LIN {X 0,Y 481.377,Z 604.114,A -85,B 0,C 180,E1 -6920.97,E2 -6920.97} C_VEL
LIN {X 0,Y 481.208,Z 611.494,A -85,B 0,C 180,E1 -6922.236,E2 -6922.236} C_VEL
LIN {X 0,Y 481.101,Z 618.078,A -85,B 0,C 180,E1 -6923.67,E2 -6923.67} C_VEL
LIN {X 0,Y 481.076,Z 622.704,A -85,B 0,C 180,E1 -6924.971,E2 -6924.971} C_VEL
LIN {X 0,Y 481.102,Z 625.077,A -85,B 0,C 180,E1 -6925.811,E2 -6925.811} C_VEL
LIN {X 0,Y 481.058,Z 626.993,A -85,B 0,C 180,E1 -6926.65,E2 -6926.65} C_VEL
LIN {X 0,Y 481.036,Z 628.433,A -85,B 0,C 180,E1 -6927.488,E2 -6927.488} C_VEL
LIN {X 0,Y 481.062,Z 630.096,A -85,B 0,C 180,E1 -6929.163,E2 -6929.163} C_VEL
LIN {X 0,Y 481.049,Z 630.319,A -85,B 0,C 180,E1 -6930,E2 -6930} C_VEL
LIN {X 0,Y 481.062,Z 630.101,A -85,B 0,C 180,E1 -6930.837,E2 -6930.837} C_VEL
LIN {X 0,Y 481.035,Z 628.45,A -85,B 0,C 180,E1 -6932.512,E2 -6932.512} C_VEL
LIN {X 0,Y 481.056,Z 627.015,A -85,B 0,C 180,E1 -6933.35,E2 -6933.35} C_VEL
LIN {X 0,Y 481.046,Z 623.991,A -85,B 0,C 180,E1 -6934.609,E2 -6934.609} C_VEL
LIN {X 0,Y 481.125,Z 619.912,A -85,B 0,C 180,E1 -6935.869,E2 -6935.869} C_VEL
LIN {X 0,Y 481.153,Z 613.626,A -85,B 0,C 180,E1 -6937.343,E2 -6937.343} C_VEL
LIN {X 0,Y 481.309,Z 606.787,A -85,B 0,C 180,E1 -6938.608,E2 -6938.608} C_VEL
LIN {X 0,Y 481.523,Z 598.317,A -85,B 0,C 180,E1 -6939.875,E2 -6939.875} C_VEL
LIN {X 0,Y 481.865,Z 589.664,A -85,B 0,C 180,E1 -6940.93,E2 -6940.93} C_VEL
LIN {X 0,Y 482.304,Z 579.305,A -85,B 0,C 180,E1 -6941.958,E2 -6941.958} C_VEL
LIN {X 0,Y 482.668,Z 568.475,A -85,B 0,C 180,E1 -6942.829,E2 -6942.829} C_VEL
LIN {X 0,Y 483.085,Z 556.965,A -85,B 0,C 180,E1 -6943.567,E2 -6943.567} C_VEL
LIN {X 0,Y 483.501,Z 545.184,A -85,B 0,C 180,E1 -6944.145,E2 -6944.145} C_VEL
LIN {X 0,Y 483.517,Z 538.3,A -85,B 0,C 180,E1 -6944.413,E2 -6944.413} C_VEL
LIN {X 0,Y 482.293,Z 527.392,A -85,B 0,C 180,E1 -6944.774,E2 -6944.774} C_VEL
LIN {X 0,Y 481.44,Z 518.405,A -85,B 0,C 180,E1 -6944.99,E2 -6944.99} C_VEL
LIN {X 0,Y 481.705,Z 503.738,A -85,B 0,C 180,E1 -6948.169,E2 -6948.169} C_VEL
LIN {X 0,Y 481.993,Z 488.984,A -85,B 0,C 180,E1 -6951.378,E2 -6951.378} C_VEL
LIN {X 0,Y 482.327,Z 474.573,A -85,B 0,C 180,E1 -6954.536,E2 -6954.536} C_VEL
LIN {X 0,Y 482.614,Z 461.951,A -85,B 0,C 180,E1 -6957.339,E2 -6957.339} C_VEL
LIN {X 0,Y 482.979,Z 449.607,A -85,B 0,C 180,E1 -6960.134,E2 -6960.134} C_VEL
LIN {X 0,Y 483.414,Z 436.079,A -85,B 0,C 180,E1 -6963.286,E2 -6963.286} C_VEL
LIN {X 0,Y 483.897,Z 423.674,A -85,B 0,C 180,E1 -6966.288,E2 -6966.288} C_VEL
LIN {X 0,Y 482.493,Z 415.613,A -85,B 0,C 180,E1 -6968.425,E2 -6968.425} C_VEL
LIN {X 0,Y 481.728,Z 411.479,A -85,B 0,C 180,E1 -6969.609,E2 -6969.609} C_VEL
LIN {X 0,Y 481.644,Z 411.493,A -85,B 0,C 180,E1 -6973.148,E2 -6973.148} C_VEL
LIN {X 0,Y 481.66,Z 411.49,A -85,B 0,C 180,E1 -6975.641,E2 -6975.641} C_VEL
LIN {X 0,Y 481.664,Z 411.488,A -85,B 0,C 180,E1 -6978.959,E2 -6978.959} C_VEL
LIN {X 0,Y 481.658,Z 411.49,A -85,B 0,C 180,E1 -6981.992,E2 -6981.992} C_VEL
LIN {X 0,Y 481.693,Z 411.483,A -85,B 0,C 180,E1 -6985.318,E2 -6985.318} C_VEL
LIN {X 0,Y 481.646,Z 411.491,A -85,B 0,C 180,E1 -6988.312,E2 -6988.312} C_VEL
LIN {X 0,Y 481.702,Z 411.482,A -85,B 0,C 180,E1 -6991.219,E2 -6991.219} C_VEL
LIN {X 0,Y 481.708,Z 411.484,A -85,B 0,C 180,E1 -6994.043,E2 -6994.043} C_VEL
LIN {X 0,Y 481.676,Z 411.486,A -85,B 0,C 180,E1 -6996.812,E2 -6996.812} C_VEL
LIN {X 0,Y 481.699,Z 411.483,A -85,B 0,C 180,E1 -6999.503,E2 -6999.503} C_VEL
LIN {X 0,Y 481.709,Z 411.484,A -85,B 0,C 180,E1 -7002.159,E2 -7002.159} C_VEL
LIN {X 0,Y 481.744,Z 411.479,A -85,B 0,C 180,E1 -7004.776,E2 -7004.776} C_VEL
LIN {X 0,Y 481.797,Z 411.474,A -85,B 0,C 180,E1 -7008.216,E2 -7008.216} C_VEL
LIN {X 0,Y 481.742,Z 411.479,A -85,B 0,C 180,E1 -7011.611,E2 -7011.611} C_VEL
LIN {X 0,Y 481.819,Z 411.47,A -85,B 0,C 180,E1 -7014.14,E2 -7014.14} C_VEL
LIN {X 0,Y 481.932,Z 411.455,A -85,B 0,C 180,E1 -7017.493,E2 -7017.493} C_VEL
LIN {X 0,Y 481.909,Z 411.457,A -85,B 0,C 180,E1 -7020.836,E2 -7020.836} C_VEL
LIN {X 0,Y 481.929,Z 411.455,A -85,B 0,C 180,E1 -7022.508,E2 -7022.508} C_VEL
LIN {X 0,Y 481.818,Z 411.471,A -85,B 0,C 180,E1 -7025.861,E2 -7025.861} C_VEL
LIN {X 0,Y 481.766,Z 411.476,A -85,B 0,C 180,E1 -7028.388,E2 -7028.388} C_VEL
LIN {X 0,Y 481.753,Z 411.478,A -85,B 0,C 180,E1 -7031.785,E2 -7031.785} C_VEL
LIN {X 0,Y 481.745,Z 411.477,A -85,B 0,C 180,E1 -7035.224,E2 -7035.224} C_VEL
LIN {X 0,Y 481.715,Z 411.481,A -85,B 0,C 180,E1 -7038.722,E2 -7038.722} C_VEL
LIN {X 0,Y 481.65,Z 411.49,A -85,B 0,C 180,E1 -7041.395,E2 -7041.395} C_VEL
LIN {X 0,Y 481.68,Z 411.488,A -85,B 0,C 180,E1 -7044.113,E2 -7044.113} C_VEL
LIN {X 0,Y 481.749,Z 411.477,A -85,B 0,C 180,E1 -7047.139,E2 -7047.139} C_VEL
LIN {X 0,Y 481.681,Z 411.488,A -85,B 0,C 180,E1 -7049.741,E2 -7049.741} C_VEL
LIN {X 0,Y 481.675,Z 411.486,A -85,B 0,C 180,E1 -7052.674,E2 -7052.674} C_VEL
LIN {X 0,Y 481.645,Z 411.492,A -85,B 0,C 180,E1 -7055.709,E2 -7055.709} C_VEL
LIN {X 0,Y 481.673,Z 411.486,A -85,B 0,C 180,E1 -7058.859,E2 -7058.859} C_VEL
LIN {X 0,Y 481.665,Z 411.489,A -85,B 0,C 180,E1 -7061.914,E2 -7061.914} C_VEL
LIN {X 0,Y 481.663,Z 411.489,A -85,B 0,C 180,E1 -7064.457,E2 -7064.457} C_VEL
LIN {X 0,Y 481.657,Z 411.492,A -85,B 0,C 180,E1 -7067.84,E2 -7067.84} C_VEL
LIN {X 0,Y 481.684,Z 411.485,A -85,B 0,C 180,E1 -7070.651,E2 -7070.651} C_VEL
LIN {X 0,Y 481.634,Z 411.493,A -85,B 0,C 180,E1 -7073.376,E2 -7073.376} C_VEL
LIN {X 0,Y 481.713,Z 411.483,A -85,B 0,C 180,E1 -7076.33,E2 -7076.33} C_VEL
LIN {X 0,Y 481.663,Z 411.489,A -85,B 0,C 180,E1 -7079.416,E2 -7079.416} C_VEL
LIN {X 0,Y 481.705,Z 411.483,A -85,B 0,C 180,E1 -7082.168,E2 -7082.168} C_VEL
LIN {X 0,Y 481.721,Z 411.48,A -85,B 0,C 180,E1 -7084.97,E2 -7084.97} C_VEL
LIN {X 0,Y 481.64,Z 411.49,A -85,B 0,C 180,E1 -7087.985,E2 -7087.985} C_VEL
LIN {X 0,Y 480.972,Z 411.574,A -85,B 0,C 180,E1 -7088.683,E2 -7088.683} C_VEL
LIN {X 0,Y 478.146,Z 411.927,A -85,B 0,C 180,E1 -7089.817,E2 -7089.817} C_VEL
LIN {X 0,Y 475.762,Z 412.224,A -85,B 0,C 180,E1 -7090.732,E2 -7090.732} C_VEL
LIN {X 0,Y 474.742,Z 412.351,A -85,B 0,C 180,E1 -7091.437,E2 -7091.437} C_VEL
LIN {X 0,Y 474.66,Z 412.361,A -85,B 0,C 180,E1 -7091.676,E2 -7091.676} C_VEL
LIN {X 0,Y 474.705,Z 412.355,A -85,B 0,C 180,E1 -7094.545,E2 -7094.545} C_VEL
LIN {X 0,Y 474.709,Z 412.354,A -85,B 0,C 180,E1 -7098.038,E2 -7098.038} C_VEL
LIN {X 0,Y 474.762,Z 412.348,A -85,B 0,C 180,E1 -7098.689,E2 -7098.689} C_VEL
LIN {X 0,Y 477.209,Z 421.926,A -85,B 0,C 180,E1 -7099.285,E2 -7099.285} C_VEL
LIN {X 0,Y 476.901,Z 433.183,A -85,B 0,C 180,E1 -7100.029,E2 -7100.029} C_VEL
LIN {X 0,Y 476.389,Z 444.579,A -85,B 0,C 180,E1 -7100.982,E2 -7100.982} C_VEL
LIN {X 0,Y 475.996,Z 453.528,A -85,B 0,C 180,E1 -7101.913,E2 -7101.913} C_VEL
LIN {X 0,Y 475.625,Z 462.093,A -85,B 0,C 180,E1 -7102.998,E2 -7102.998} C_VEL
LIN {X 0,Y 475.251,Z 470.197,A -85,B 0,C 180,E1 -7104.271,E2 -7104.271} C_VEL
LIN {X 0,Y 474.95,Z 475.754,A -85,B 0,C 180,E1 -7105.332,E2 -7105.332} C_VEL
LIN {X 0,Y 474.707,Z 481.159,A -85,B 0,C 180,E1 -7106.605,E2 -7106.605} C_VEL
LIN {X 0,Y 474.572,Z 485.4,A -85,B 0,C 180,E1 -7107.878,E2 -7107.878} C_VEL
LIN {X 0,Y 474.352,Z 488.628,A -85,B 0,C 180,E1 -7109.151,E2 -7109.151} C_VEL
LIN {X 0,Y 474.295,Z 490.225,A -85,B 0,C 180,E1 -7110,E2 -7110} C_VEL
LIN {X 0,Y 474.172,Z 491.447,A -85,B 0,C 180,E1 -7110.849,E2 -7110.849} C_VEL
LIN {X 0,Y 474.232,Z 492.256,A -85,B 0,C 180,E1 -7111.699,E2 -7111.699} C_VEL
LIN {X 0,Y 474.206,Z 492.692,A -85,B 0,C 180,E1 -7113.399,E2 -7113.399} C_VEL
LIN {X 0,Y 474.321,Z 491.624,A -85,B 0,C 180,E1 -7115.101,E2 -7115.101} C_VEL
LIN {X 0,Y 474.401,Z 488.934,A -85,B 0,C 180,E1 -7116.807,E2 -7116.807} C_VEL
LIN {X 0,Y 474.522,Z 485.822,A -85,B 0,C 180,E1 -7118.089,E2 -7118.089} C_VEL
LIN {X 0,Y 474.749,Z 481.653,A -85,B 0,C 180,E1 -7119.372,E2 -7119.372} C_VEL
LIN {X 0,Y 475.063,Z 475.32,A -85,B 0,C 180,E1 -7120.873,E2 -7120.873} C_VEL
LIN {X 0,Y 475.337,Z 468.074,A -85,B 0,C 180,E1 -7122.206,E2 -7122.206} C_VEL
LIN {X 0,Y 475.767,Z 459.593,A -85,B 0,C 180,E1 -7123.454,E2 -7123.454} C_VEL
LIN {X 0,Y 476.167,Z 450.586,A -85,B 0,C 180,E1 -7124.532,E2 -7124.532} C_VEL
LIN {X 0,Y 476.623,Z 440.519,A -85,B 0,C 180,E1 -7125.502,E2 -7125.502} C_VEL
LIN {X 0,Y 477.01,Z 429.745,A -85,B 0,C 180,E1 -7126.335,E2 -7126.335} C_VEL
LIN {X 0,Y 477.127,Z 420.99,A -85,B 0,C 180,E1 -7126.89,E2 -7126.89} C_VEL
LIN {X 0,Y 474.656,Z 412.36,A -85,B 0,C 180,E1 -7127.448,E2 -7127.448} C_VEL
LIN {X 0,Y 474.659,Z 412.361,A -85,B 0,C 180,E1 -7129.91,E2 -7129.91} C_VEL
LIN {X 0,Y 474.64,Z 412.357,A -85,B 0,C 180,E1 -7133.358,E2 -7133.358} C_VEL
LIN {X 0,Y 474.66,Z 412.362,A -85,B 0,C 180,E1 -7136.372,E2 -7136.372} C_VEL
LIN {X 0,Y 474.626,Z 412.359,A -85,B 0,C 180,E1 -7139.252,E2 -7139.252} C_VEL
LIN {X 0,Y 474.62,Z 412.365,A -85,B 0,C 180,E1 -7142.431,E2 -7142.431} C_VEL
LIN {X 0,Y 474.624,Z 412.36,A -85,B 0,C 180,E1 -7145.47,E2 -7145.47} C_VEL
LIN {X 0,Y 474.617,Z 412.364,A -85,B 0,C 180,E1 -7148.457,E2 -7148.457} C_VEL
LIN {X 0,Y 474.632,Z 412.358,A -85,B 0,C 180,E1 -7150.959,E2 -7150.959} C_VEL
LIN {X 0,Y 474.614,Z 412.369,A -85,B 0,C 180,E1 -7154.105,E2 -7154.105} C_VEL
LIN {X 0,Y 474.62,Z 412.359,A -85,B 0,C 180,E1 -7157.066,E2 -7157.066} C_VEL
LIN {X 0,Y 474.649,Z 412.358,A -85,B 0,C 180,E1 -7160.454,E2 -7160.454} C_VEL
LIN {X 0,Y 474.593,Z 412.367,A -85,B 0,C 180,E1 -7163.676,E2 -7163.676} C_VEL
LIN {X 0,Y 474.647,Z 412.356,A -85,B 0,C 180,E1 -7166.78,E2 -7166.78} C_VEL
LIN {X 0,Y 474.61,Z 412.367,A -85,B 0,C 180,E1 -7169.77,E2 -7169.77} C_VEL
LIN {X 0,Y 474.702,Z 412.349,A -85,B 0,C 180,E1 -7172.68,E2 -7172.68} C_VEL
LIN {X 0,Y 474.645,Z 412.36,A -85,B 0,C 180,E1 -7175.506,E2 -7175.506} C_VEL
LIN {X 0,Y 474.675,Z 412.354,A -85,B 0,C 180,E1 -7179.185,E2 -7179.185} C_VEL
LIN {X 0,Y 474.651,Z 412.362,A -85,B 0,C 180,E1 -7181.884,E2 -7181.884} C_VEL
LIN {X 0,Y 474.704,Z 412.349,A -85,B 0,C 180,E1 -7184.544,E2 -7184.544} C_VEL
LIN {X 0,Y 474.662,Z 412.358,A -85,B 0,C 180,E1 -7186.874,E2 -7186.874} C_VEL
LIN {X 0,Y 476.753,Z 420.106,A -85,B 0,C 180,E1 -7187.367,E2 -7187.367} C_VEL
LIN {X 0,Y 476.502,Z 430.082,A -85,B 0,C 180,E1 -7188.007,E2 -7188.007} C_VEL
LIN {X 0,Y 476.131,Z 441.708,A -85,B 0,C 180,E1 -7188.937,E2 -7188.937} C_VEL
LIN {X 0,Y 475.81,Z 450.358,A -85,B 0,C 180,E1 -7189.79,E2 -7189.79} C_VEL
LIN {X 0,Y 475.421,Z 459.298,A -85,B 0,C 180,E1 -7190.856,E2 -7190.856} C_VEL
LIN {X 0,Y 475.084,Z 468.019,A -85,B 0,C 180,E1 -7192.135,E2 -7192.135} C_VEL
LIN {X 0,Y 474.872,Z 475.039,A -85,B 0,C 180,E1 -7193.414,E2 -7193.414} C_VEL
LIN {X 0,Y 474.479,Z 481.448,A -85,B 0,C 180,E1 -7194.901,E2 -7194.901} C_VEL
LIN {X 0,Y 474.487,Z 485.65,A -85,B 0,C 180,E1 -7196.178,E2 -7196.178} C_VEL
LIN {X 0,Y 474.218,Z 488.842,A -85,B 0,C 180,E1 -7197.452,E2 -7197.452} C_VEL
LIN {X 0,Y 474.242,Z 490.427,A -85,B 0,C 180,E1 -7198.301,E2 -7198.301} C_VEL
LIN {X 0,Y 474.17,Z 491.584,A -85,B 0,C 180,E1 -7199.151,E2 -7199.151} C_VEL
LIN {X 0,Y 474.167,Z 492.694,A -85,B 0,C 180,E1 -7200.849,E2 -7200.849} C_VEL
LIN {X 0,Y 474.232,Z 492.669,A -85,B 0,C 180,E1 -7201.698,E2 -7201.698} C_VEL
LIN {X 0,Y 474.263,Z 491.378,A -85,B 0,C 180,E1 -7203.398,E2 -7203.398} C_VEL
LIN {X 0,Y 474.329,Z 490.156,A -85,B 0,C 180,E1 -7204.248,E2 -7204.248} C_VEL
LIN {X 0,Y 474.483,Z 487.49,A -85,B 0,C 180,E1 -7205.525,E2 -7205.525} C_VEL
LIN {X 0,Y 474.665,Z 483.805,A -85,B 0,C 180,E1 -7206.803,E2 -7206.803} C_VEL
LIN {X 0,Y 474.832,Z 478.985,A -85,B 0,C 180,E1 -7208.083,E2 -7208.083} C_VEL
LIN {X 0,Y 475.145,Z 472.826,A -85,B 0,C 180,E1 -7209.364,E2 -7209.364} C_VEL
LIN {X 0,Y 475.462,Z 465.142,A -85,B 0,C 180,E1 -7210.648,E2 -7210.648} C_VEL
LIN {X 0,Y 475.809,Z 457.258,A -85,B 0,C 180,E1 -7211.718,E2 -7211.718} C_VEL
LIN {X 0,Y 476.148,Z 447.587,A -85,B 0,C 180,E1 -7212.791,E2 -7212.791} C_VEL
LIN {X 0,Y 476.651,Z 436.734,A -85,B 0,C 180,E1 -7213.754,E2 -7213.754} C_VEL
LIN {X 0,Y 477.028,Z 426.184,A -85,B 0,C 180,E1 -7214.505,E2 -7214.505} C_VEL
LIN {X 0,Y 476.99,Z 420.79,A -85,B 0,C 180,E1 -7214.833,E2 -7214.833} C_VEL
LIN {X 0,Y 474.697,Z 412.357,A -85,B 0,C 180,E1 -7215.373,E2 -7215.373} C_VEL
LIN {X 0,Y 474.663,Z 412.366,A -85,B 0,C 180,E1 -7218.629,E2 -7218.629} C_VEL
LIN {X 0,Y 474.639,Z 412.367,A -85,B 0,C 180,E1 -7221.116,E2 -7221.116} C_VEL
LIN {X 0,Y 474.644,Z 412.363,A -85,B 0,C 180,E1 -7224.494,E2 -7224.494} C_VEL
LIN {X 0,Y 474.703,Z 412.355,A -85,B 0,C 180,E1 -7227.338,E2 -7227.338} C_VEL
LIN {X 0,Y 474.608,Z 412.367,A -85,B 0,C 180,E1 -7230.81,E2 -7230.81} C_VEL
LIN {X 0,Y 474.641,Z 412.363,A -85,B 0,C 180,E1 -7233.984,E2 -7233.984} C_VEL
LIN {X 0,Y 474.575,Z 412.372,A -85,B 0,C 180,E1 -7236.899,E2 -7236.899} C_VEL
LIN {X 0,Y 474.63,Z 412.364,A -85,B 0,C 180,E1 -7239.647,E2 -7239.647} C_VEL
LIN {X 0,Y 474.618,Z 412.366,A -85,B 0,C 180,E1 -7242.934,E2 -7242.934} C_VEL
LIN {X 0,Y 474.612,Z 412.364,A -85,B 0,C 180,E1 -7245.895,E2 -7245.895} C_VEL
LIN {X 0,Y 474.631,Z 412.364,A -85,B 0,C 180,E1 -7249.041,E2 -7249.041} C_VEL
LIN {X 0,Y 474.67,Z 412.558,A -85,B 0,C 180,E1 -7249.868,E2 -7249.868} C_VEL
LIN {X 0,Y 476.752,Z 422.929,A -85,B 0,C 180,E1 -7252.814,E2 -7252.814} C_VEL
LIN {X 0,Y 477.156,Z 426.977,A -85,B 0,C 180,E1 -7253.902,E2 -7253.902} C_VEL
LIN {X 0,Y 476.36,Z 441.74,A -85,B 0,C 180,E1 -7257.572,E2 -7257.572} C_VEL
LIN {X 0,Y 475.905,Z 454.457,A -85,B 0,C 180,E1 -7260.609,E2 -7260.609} C_VEL
LIN {X 0,Y 475.492,Z 467.701,A -85,B 0,C 180,E1 -7263.678,E2 -7263.678} C_VEL
LIN {X 0,Y 475.158,Z 480.12,A -85,B 0,C 180,E1 -7266.497,E2 -7266.497} C_VEL
LIN {X 0,Y 474.78,Z 494.181,A -85,B 0,C 180,E1 -7269.643,E2 -7269.643} C_VEL
LIN {X 0,Y 474.542,Z 508.253,A -85,B 0,C 180,E1 -7272.77,E2 -7272.77} C_VEL
LIN {X 0,Y 474.368,Z 517.338,A -85,B 0,C 180,E1 -7274.781,E2 -7274.781} C_VEL
LIN {X 0,Y 475.741,Z 532.276,A -85,B 0,C 180,E1 -7275.182,E2 -7275.182} C_VEL
LIN {X 0,Y 476.7,Z 541.484,A -85,B 0,C 180,E1 -7275.539,E2 -7275.539} C_VEL
LIN {X 0,Y 476.207,Z 553.915,A -85,B 0,C 180,E1 -7276.124,E2 -7276.124} C_VEL
LIN {X 0,Y 475.712,Z 565.91,A -85,B 0,C 180,E1 -7276.871,E2 -7276.871} C_VEL
LIN {X 0,Y 475.293,Z 576.474,A -85,B 0,C 180,E1 -7277.707,E2 -7277.707} C_VEL
LIN {X 0,Y 474.861,Z 586.571,A -85,B 0,C 180,E1 -7278.691,E2 -7278.691} C_VEL
LIN {X 0,Y 474.527,Z 595.599,A -85,B 0,C 180,E1 -7279.762,E2 -7279.762} C_VEL
LIN {X 0,Y 474.265,Z 604.436,A -85,B 0,C 180,E1 -7281.048,E2 -7281.048} C_VEL
LIN {X 0,Y 474.108,Z 611.516,A -85,B 0,C 180,E1 -7282.333,E2 -7282.333} C_VEL
LIN {X 0,Y 474.037,Z 617.39,A -85,B 0,C 180,E1 -7283.663,E2 -7283.663} C_VEL
LIN {X 0,Y 474.03,Z 621.682,A -85,B 0,C 180,E1 -7284.896,E2 -7284.896} C_VEL
LIN {X 0,Y 474.036,Z 624.054,A -85,B 0,C 180,E1 -7285.749,E2 -7285.749} C_VEL
LIN {X 0,Y 474.013,Z 625.974,A -85,B 0,C 180,E1 -7286.6,E2 -7286.6} C_VEL
LIN {X 0,Y 473.997,Z 627.416,A -85,B 0,C 180,E1 -7287.45,E2 -7287.45} C_VEL
LIN {X 0,Y 474.051,Z 629.086,A -85,B 0,C 180,E1 -7289.15,E2 -7289.15} C_VEL
LIN {X 0,Y 474.036,Z 629.31,A -85,B 0,C 180,E1 -7290,E2 -7290} C_VEL
LIN {X 0,Y 474.05,Z 629.092,A -85,B 0,C 180,E1 -7290.849,E2 -7290.849} C_VEL
LIN {X 0,Y 473.995,Z 627.437,A -85,B 0,C 180,E1 -7292.549,E2 -7292.549} C_VEL
LIN {X 0,Y 474.01,Z 626,A -85,B 0,C 180,E1 -7293.4,E2 -7293.4} C_VEL
LIN {X 0,Y 474.001,Z 622.976,A -85,B 0,C 180,E1 -7294.677,E2 -7294.677} C_VEL
LIN {X 0,Y 474.06,Z 618.892,A -85,B 0,C 180,E1 -7295.956,E2 -7295.956} C_VEL
LIN {X 0,Y 474.099,Z 612.606,A -85,B 0,C 180,E1 -7297.453,E2 -7297.453} C_VEL
LIN {X 0,Y 474.236,Z 605.761,A -85,B 0,C 180,E1 -7298.737,E2 -7298.737} C_VEL
LIN {X 0,Y 474.476,Z 597.292,A -85,B 0,C 180,E1 -7300.023,E2 -7300.023} C_VEL
LIN {X 0,Y 474.825,Z 588.636,A -85,B 0,C 180,E1 -7301.094,E2 -7301.094} C_VEL
LIN {X 0,Y 475.291,Z 578.561,A -85,B 0,C 180,E1 -7302.111,E2 -7302.111} C_VEL
LIN {X 0,Y 475.623,Z 568.892,A -85,B 0,C 180,E1 -7302.914,E2 -7302.914} C_VEL
LIN {X 0,Y 476.068,Z 557.722,A -85,B 0,C 180,E1 -7303.662,E2 -7303.662} C_VEL
LIN {X 0,Y 476.527,Z 545.375,A -85,B 0,C 180,E1 -7304.302,E2 -7304.302} C_VEL
LIN {X 0,Y 476.475,Z 538.387,A -85,B 0,C 180,E1 -7304.59,E2 -7304.59} C_VEL
LIN {X 0,Y 475.375,Z 527.969,A -85,B 0,C 180,E1 -7304.953,E2 -7304.953} C_VEL
LIN {X 0,Y 474.368,Z 517.419,A -85,B 0,C 180,E1 -7305.219,E2 -7305.219} C_VEL
LIN {X 0,Y 474.635,Z 503.154,A -85,B 0,C 180,E1 -7308.367,E2 -7308.367} C_VEL
LIN {X 0,Y 474.953,Z 488.049,A -85,B 0,C 180,E1 -7311.711,E2 -7311.711} C_VEL
LIN {X 0,Y 475.318,Z 473.658,A -85,B 0,C 180,E1 -7314.923,E2 -7314.923} C_VEL
LIN {X 0,Y 475.694,Z 459.14,A -85,B 0,C 180,E1 -7318.214,E2 -7318.214} C_VEL
LIN {X 0,Y 476.092,Z 446.662,A -85,B 0,C 180,E1 -7321.109,E2 -7321.109} C_VEL
LIN {X 0,Y 476.603,Z 433.186,A -85,B 0,C 180,E1 -7324.332,E2 -7324.332} C_VEL
LIN {X 0,Y 476.938,Z 424.934,A -85,B 0,C 180,E1 -7326.376,E2 -7326.376} C_VEL
LIN {X 0,Y 475.59,Z 417.265,A -85,B 0,C 180,E1 -7328.445,E2 -7328.445} C_VEL
LIN {X 0,Y 474.696,Z 412.356,A -85,B 0,C 180,E1 -7329.849,E2 -7329.849} C_VEL
LIN {X 0,Y 474.616,Z 412.369,A -85,B 0,C 180,E1 -7332.934,E2 -7332.934} C_VEL
LIN {X 0,Y 474.616,Z 412.368,A -85,B 0,C 180,E1 -7335.896,E2 -7335.896} C_VEL
LIN {X 0,Y 474.633,Z 412.363,A -85,B 0,C 180,E1 -7339.04,E2 -7339.04} C_VEL
LIN {X 0,Y 474.612,Z 412.367,A -85,B 0,C 180,E1 -7341.704,E2 -7341.704} C_VEL
LIN {X 0,Y 474.63,Z 412.364,A -85,B 0,C 180,E1 -7344.726,E2 -7344.726} C_VEL
LIN {X 0,Y 474.636,Z 412.364,A -85,B 0,C 180,E1 -7347.788,E2 -7347.788} C_VEL
LIN {X 0,Y 474.625,Z 412.365,A -85,B 0,C 180,E1 -7350.884,E2 -7350.884} C_VEL
LIN {X 0,Y 474.668,Z 412.36,A -85,B 0,C 180,E1 -7353.629,E2 -7353.629} C_VEL
LIN {X 0,Y 474.637,Z 412.363,A -85,B 0,C 180,E1 -7356.641,E2 -7356.641} C_VEL
LIN {X 0,Y 474.658,Z 412.362,A -85,B 0,C 180,E1 -7360.09,E2 -7360.09} C_VEL
LIN {X 0,Y 474.653,Z 412.361,A -85,B 0,C 180,E1 -7362.775,E2 -7362.775} C_VEL
LIN {X 0,Y 474.65,Z 412.362,A -85,B 0,C 180,E1 -7365.421,E2 -7365.421} C_VEL
LIN {X 0,Y 474.741,Z 412.352,A -85,B 0,C 180,E1 -7368.039,E2 -7368.039} C_VEL
LIN {X 0,Y 474.714,Z 412.353,A -85,B 0,C 180,E1 -7371.486,E2 -7371.486} C_VEL
LIN {X 0,Y 474.781,Z 412.347,A -85,B 0,C 180,E1 -7374.053,E2 -7374.053} C_VEL
LIN {X 0,Y 474.898,Z 412.331,A -85,B 0,C 180,E1 -7377.456,E2 -7377.456} C_VEL
LIN {X 0,Y 474.914,Z 412.33,A -85,B 0,C 180,E1 -7380,E2 -7380} C_VEL
LIN {X 0,Y 474.895,Z 412.331,A -85,B 0,C 180,E1 -7382.545,E2 -7382.545} C_VEL
LIN {X 0,Y 474.781,Z 412.347,A -85,B 0,C 180,E1 -7385.948,E2 -7385.948} C_VEL
LIN {X 0,Y 474.731,Z 412.353,A -85,B 0,C 180,E1 -7388.514,E2 -7388.514} C_VEL
LIN {X 0,Y 474.707,Z 412.357,A -85,B 0,C 180,E1 -7391.963,E2 -7391.963} C_VEL
LIN {X 0,Y 474.702,Z 412.356,A -85,B 0,C 180,E1 -7395.456,E2 -7395.456} C_VEL
LIN {X 0,Y 474.668,Z 412.358,A -85,B 0,C 180,E1 -7399.01,E2 -7399.01} C_VEL
LIN {X 0,Y 474.593,Z 412.37,A -85,B 0,C 180,E1 -7401.729,E2 -7401.729} C_VEL
LIN {X 0,Y 474.662,Z 412.36,A -85,B 0,C 180,E1 -7404.493,E2 -7404.493} C_VEL
LIN {X 0,Y 474.701,Z 412.355,A -85,B 0,C 180,E1 -7407.339,E2 -7407.339} C_VEL
LIN {X 0,Y 474.607,Z 412.366,A -85,B 0,C 180,E1 -7410.81,E2 -7410.81} C_VEL
LIN {X 0,Y 474.641,Z 412.364,A -85,B 0,C 180,E1 -7413.984,E2 -7413.984} C_VEL
LIN {X 0,Y 474.577,Z 412.37,A -85,B 0,C 180,E1 -7416.9,E2 -7416.9} C_VEL
LIN {X 0,Y 474.63,Z 412.365,A -85,B 0,C 180,E1 -7419.648,E2 -7419.648} C_VEL
LIN {X 0,Y 474.638,Z 412.362,A -85,B 0,C 180,E1 -7422.932,E2 -7422.932} C_VEL
LIN {X 0,Y 474.618,Z 412.367,A -85,B 0,C 180,E1 -7425.896,E2 -7425.896} C_VEL
LIN {X 0,Y 474.635,Z 412.363,A -85,B 0,C 180,E1 -7429.04,E2 -7429.04} C_VEL
LIN {X 0,Y 474.614,Z 412.367,A -85,B 0,C 180,E1 -7431.704,E2 -7431.704} C_VEL
LIN {X 0,Y 474.633,Z 412.362,A -85,B 0,C 180,E1 -7434.726,E2 -7434.726} C_VEL
LIN {X 0,Y 474.642,Z 412.364,A -85,B 0,C 180,E1 -7437.788,E2 -7437.788} C_VEL
LIN {X 0,Y 474.635,Z 412.363,A -85,B 0,C 180,E1 -7440.883,E2 -7440.883} C_VEL
LIN {X 0,Y 474.665,Z 412.361,A -85,B 0,C 180,E1 -7443.629,E2 -7443.629} C_VEL
LIN {X 0,Y 474.639,Z 412.361,A -85,B 0,C 180,E1 -7446.642,E2 -7446.642} C_VEL
LIN {X 0,Y 474.661,Z 412.361,A -85,B 0,C 180,E1 -7450.09,E2 -7450.09} C_VEL
LIN {X 0,Y 474.66,Z 412.361,A -85,B 0,C 180,E1 -7451.676,E2 -7451.676} C_VEL
LIN {X 0,Y 473.997,Z 412.445,A -85,B 0,C 180,E1 -7452.385,E2 -7452.385} C_VEL
LIN {X 0,Y 471.146,Z 412.802,A -85,B 0,C 180,E1 -7453.537,E2 -7453.537} C_VEL
LIN {X 0,Y 468.73,Z 413.102,A -85,B 0,C 180,E1 -7454.465,E2 -7454.465} C_VEL
LIN {X 0,Y 467.688,Z 413.23,A -85,B 0,C 180,E1 -7455.182,E2 -7455.182} C_VEL
LIN {X 0,Y 467.601,Z 413.24,A -85,B 0,C 180,E1 -7455.425,E2 -7455.425} C_VEL
LIN {X 0,Y 467.7,Z 413.229,A -85,B 0,C 180,E1 -7458.461,E2 -7458.461} C_VEL
LIN {X 0,Y 470.351,Z 423.533,A -85,B 0,C 180,E1 -7459.127,E2 -7459.127} C_VEL
LIN {X 0,Y 470.022,Z 434.663,A -85,B 0,C 180,E1 -7459.881,E2 -7459.881} C_VEL
LIN {X 0,Y 469.489,Z 445.977,A -85,B 0,C 180,E1 -7460.849,E2 -7460.849} C_VEL
LIN {X 0,Y 469.083,Z 454.859,A -85,B 0,C 180,E1 -7461.793,E2 -7461.793} C_VEL
LIN {X 0,Y 468.673,Z 463.358,A -85,B 0,C 180,E1 -7462.894,E2 -7462.894} C_VEL
LIN {X 0,Y 468.294,Z 471.413,A -85,B 0,C 180,E1 -7464.186,E2 -7464.186} C_VEL
LIN {X 0,Y 467.97,Z 476.934,A -85,B 0,C 180,E1 -7465.262,E2 -7465.262} C_VEL
LIN {X 0,Y 467.716,Z 482.305,A -85,B 0,C 180,E1 -7466.554,E2 -7466.554} C_VEL
LIN {X 0,Y 467.575,Z 486.515,A -85,B 0,C 180,E1 -7467.847,E2 -7467.847} C_VEL
LIN {X 0,Y 467.345,Z 489.714,A -85,B 0,C 180,E1 -7469.139,E2 -7469.139} C_VEL
LIN {X 0,Y 467.285,Z 491.297,A -85,B 0,C 180,E1 -7470,E2 -7470} C_VEL
LIN {X 0,Y 467.153,Z 492.507,A -85,B 0,C 180,E1 -7470.862,E2 -7470.862} C_VEL
LIN {X 0,Y 467.216,Z 493.29,A -85,B 0,C 180,E1 -7471.724,E2 -7471.724} C_VEL
LIN {X 0,Y 467.18,Z 493.698,A -85,B 0,C 180,E1 -7473.45,E2 -7473.45} C_VEL
LIN {X 0,Y 467.316,Z 492.591,A -85,B 0,C 180,E1 -7475.177,E2 -7475.177} C_VEL
LIN {X 0,Y 467.423,Z 489.867,A -85,B 0,C 180,E1 -7476.909,E2 -7476.909} C_VEL
LIN {X 0,Y 467.545,Z 486.728,A -85,B 0,C 180,E1 -7478.21,E2 -7478.21} C_VEL
LIN {X 0,Y 467.795,Z 482.528,A -85,B 0,C 180,E1 -7479.513,E2 -7479.513} C_VEL
LIN {X 0,Y 468.085,Z 477.152,A -85,B 0,C 180,E1 -7480.818,E2 -7480.818} C_VEL
LIN {X 0,Y 468.317,Z 470.429,A -85,B 0,C 180,E1 -7482.128,E2 -7482.128} C_VEL
LIN {X 0,Y 468.826,Z 461.936,A -85,B 0,C 180,E1 -7483.436,E2 -7483.436} C_VEL
LIN {X 0,Y 469.243,Z 453.201,A -85,B 0,C 180,E1 -7484.529,E2 -7484.529} C_VEL
LIN {X 0,Y 469.664,Z 443.563,A -85,B 0,C 180,E1 -7485.515,E2 -7485.515} C_VEL
LIN {X 0,Y 470.108,Z 432.93,A -85,B 0,C 180,E1 -7486.39,E2 -7486.39} C_VEL
LIN {X 0,Y 470.454,Z 423.015,A -85,B 0,C 180,E1 -7487.042,E2 -7487.042} C_VEL
LIN {X 0,Y 467.618,Z 413.238,A -85,B 0,C 180,E1 -7487.691,E2 -7487.691} C_VEL
LIN {X 0,Y 467.628,Z 413.238,A -85,B 0,C 180,E1 -7490.223,E2 -7490.223} C_VEL
LIN {X 0,Y 467.568,Z 413.241,A -85,B 0,C 180,E1 -7493.944,E2 -7493.944} C_VEL
LIN {X 0,Y 467.618,Z 413.234,A -85,B 0,C 180,E1 -7496.801,E2 -7496.801} C_VEL
LIN {X 0,Y 467.559,Z 413.241,A -85,B 0,C 180,E1 -7499.738,E2 -7499.738} C_VEL
LIN {X 0,Y 467.588,Z 413.237,A -85,B 0,C 180,E1 -7502.758,E2 -7502.758} C_VEL
LIN {X 0,Y 467.561,Z 413.243,A -85,B 0,C 180,E1 -7505.889,E2 -7505.889} C_VEL
LIN {X 0,Y 467.587,Z 413.236,A -85,B 0,C 180,E1 -7509.145,E2 -7509.145} C_VEL
LIN {X 0,Y 467.591,Z 413.238,A -85,B 0,C 180,E1 -7512.567,E2 -7512.567} C_VEL
LIN {X 0,Y 467.575,Z 413.237,A -85,B 0,C 180,E1 -7515.053,E2 -7515.053} C_VEL
LIN {X 0,Y 467.593,Z 413.236,A -85,B 0,C 180,E1 -7517.44,E2 -7517.44} C_VEL
LIN {X 0,Y 467.587,Z 413.236,A -85,B 0,C 180,E1 -7520.855,E2 -7520.855} C_VEL
LIN {X 0,Y 467.564,Z 413.243,A -85,B 0,C 180,E1 -7524.261,E2 -7524.261} C_VEL
LIN {X 0,Y 467.586,Z 413.237,A -85,B 0,C 180,E1 -7527.321,E2 -7527.321} C_VEL
LIN {X 0,Y 467.574,Z 413.238,A -85,B 0,C 180,E1 -7530.667,E2 -7530.667} C_VEL
LIN {X 0,Y 467.617,Z 413.233,A -85,B 0,C 180,E1 -7533.199,E2 -7533.199} C_VEL
LIN {X 0,Y 467.595,Z 413.236,A -85,B 0,C 180,E1 -7536.469,E2 -7536.469} C_VEL
LIN {X 0,Y 467.627,Z 413.239,A -85,B 0,C 180,E1 -7539.777,E2 -7539.777} C_VEL
LIN {X 0,Y 467.603,Z 413.234,A -85,B 0,C 180,E1 -7542.506,E2 -7542.506} C_VEL
LIN {X 0,Y 467.611,Z 413.235,A -85,B 0,C 180,E1 -7545.196,E2 -7545.196} C_VEL
LIN {X 0,Y 467.656,Z 413.231,A -85,B 0,C 180,E1 -7546.674,E2 -7546.674} C_VEL
LIN {X 0,Y 469.962,Z 422.285,A -85,B 0,C 180,E1 -7547.266,E2 -7547.266} C_VEL
LIN {X 0,Y 469.528,Z 433.423,A -85,B 0,C 180,E1 -7548.013,E2 -7548.013} C_VEL
LIN {X 0,Y 469.089,Z 444.801,A -85,B 0,C 180,E1 -7548.987,E2 -7548.987} C_VEL
LIN {X 0,Y 468.796,Z 454.989,A -85,B 0,C 180,E1 -7550.072,E2 -7550.072} C_VEL
LIN {X 0,Y 468.358,Z 463.311,A -85,B 0,C 180,E1 -7551.152,E2 -7551.152} C_VEL
LIN {X 0,Y 467.991,Z 471.618,A -85,B 0,C 180,E1 -7552.485,E2 -7552.485} C_VEL
LIN {X 0,Y 467.779,Z 476.961,A -85,B 0,C 180,E1 -7553.53,E2 -7553.53} C_VEL
LIN {X 0,Y 467.48,Z 482.39,A -85,B 0,C 180,E1 -7554.825,E2 -7554.825} C_VEL
LIN {X 0,Y 467.475,Z 486.614,A -85,B 0,C 180,E1 -7556.121,E2 -7556.121} C_VEL
LIN {X 0,Y 467.195,Z 489.826,A -85,B 0,C 180,E1 -7557.413,E2 -7557.413} C_VEL
LIN {X 0,Y 467.227,Z 491.421,A -85,B 0,C 180,E1 -7558.276,E2 -7558.276} C_VEL
LIN {X 0,Y 467.151,Z 492.585,A -85,B 0,C 180,E1 -7559.138,E2 -7559.138} C_VEL
LIN {X 0,Y 467.148,Z 493.713,A -85,B 0,C 180,E1 -7560.862,E2 -7560.862} C_VEL
LIN {X 0,Y 467.217,Z 493.688,A -85,B 0,C 180,E1 -7561.724,E2 -7561.724} C_VEL
LIN {X 0,Y 467.248,Z 492.406,A -85,B 0,C 180,E1 -7563.449,E2 -7563.449} C_VEL
LIN {X 0,Y 467.319,Z 491.183,A -85,B 0,C 180,E1 -7564.312,E2 -7564.312} C_VEL
LIN {X 0,Y 467.495,Z 488.51,A -85,B 0,C 180,E1 -7565.608,E2 -7565.608} C_VEL
LIN {X 0,Y 467.688,Z 484.815,A -85,B 0,C 180,E1 -7566.905,E2 -7566.905} C_VEL
LIN {X 0,Y 467.874,Z 479.981,A -85,B 0,C 180,E1 -7568.204,E2 -7568.204} C_VEL
LIN {X 0,Y 468.208,Z 473.832,A -85,B 0,C 180,E1 -7569.504,E2 -7569.504} C_VEL
LIN {X 0,Y 468.559,Z 466.164,A -85,B 0,C 180,E1 -7570.806,E2 -7570.806} C_VEL
LIN {X 0,Y 468.95,Z 458.299,A -85,B 0,C 180,E1 -7571.892,E2 -7571.892} C_VEL
LIN {X 0,Y 469.3,Z 448.613,A -85,B 0,C 180,E1 -7572.981,E2 -7572.981} C_VEL
LIN {X 0,Y 469.853,Z 437.746,A -85,B 0,C 180,E1 -7573.957,E2 -7573.957} C_VEL
LIN {X 0,Y 470.235,Z 427.169,A -85,B 0,C 180,E1 -7574.719,E2 -7574.719} C_VEL
LIN {X 0,Y 470.322,Z 423.59,A -85,B 0,C 180,E1 -7574.937,E2 -7574.937} C_VEL
LIN {X 0,Y 468.399,Z 415.775,A -85,B 0,C 180,E1 -7575.446,E2 -7575.446} C_VEL
LIN {X 0,Y 467.662,Z 413.234,A -85,B 0,C 180,E1 -7575.61,E2 -7575.61} C_VEL
LIN {X 0,Y 467.618,Z 413.244,A -85,B 0,C 180,E1 -7578.763,E2 -7578.763} C_VEL
LIN {X 0,Y 467.584,Z 413.246,A -85,B 0,C 180,E1 -7581.268,E2 -7581.268} C_VEL
LIN {X 0,Y 467.567,Z 413.245,A -85,B 0,C 180,E1 -7583.944,E2 -7583.944} C_VEL
LIN {X 0,Y 467.617,Z 413.238,A -85,B 0,C 180,E1 -7586.8,E2 -7586.8} C_VEL
LIN {X 0,Y 467.558,Z 413.245,A -85,B 0,C 180,E1 -7589.738,E2 -7589.738} C_VEL
LIN {X 0,Y 467.587,Z 413.243,A -85,B 0,C 180,E1 -7592.758,E2 -7592.758} C_VEL
LIN {X 0,Y 467.557,Z 413.246,A -85,B 0,C 180,E1 -7595.889,E2 -7595.889} C_VEL
LIN {X 0,Y 467.585,Z 413.24,A -85,B 0,C 180,E1 -7599.145,E2 -7599.145} C_VEL
LIN {X 0,Y 467.589,Z 413.243,A -85,B 0,C 180,E1 -7602.567,E2 -7602.567} C_VEL
LIN {X 0,Y 467.574,Z 413.245,A -85,B 0,C 180,E1 -7605.053,E2 -7605.053} C_VEL
LIN {X 0,Y 467.592,Z 413.241,A -85,B 0,C 180,E1 -7607.44,E2 -7607.44} C_VEL
LIN {X 0,Y 467.602,Z 413.304,A -85,B 0,C 180,E1 -7609.526,E2 -7609.526} C_VEL
LIN {X 0,Y 469.623,Z 423.492,A -85,B 0,C 180,E1 -7612.482,E2 -7612.482} C_VEL
LIN {X 0,Y 470.23,Z 428.33,A -85,B 0,C 180,E1 -7613.812,E2 -7613.812} C_VEL
LIN {X 0,Y 469.421,Z 442.433,A -85,B 0,C 180,E1 -7617.386,E2 -7617.386} C_VEL
LIN {X 0,Y 468.918,Z 454.732,A -85,B 0,C 180,E1 -7620.376,E2 -7620.376} C_VEL
LIN {X 0,Y 468.472,Z 467.929,A -85,B 0,C 180,E1 -7623.493,E2 -7623.493} C_VEL
LIN {X 0,Y 468.079,Z 481.68,A -85,B 0,C 180,E1 -7626.672,E2 -7626.672} C_VEL
LIN {X 0,Y 467.685,Z 495.314,A -85,B 0,C 180,E1 -7629.78,E2 -7629.78} C_VEL
LIN {X 0,Y 467.476,Z 507.314,A -85,B 0,C 180,E1 -7632.501,E2 -7632.501} C_VEL
LIN {X 0,Y 467.289,Z 516.403,A -85,B 0,C 180,E1 -7634.544,E2 -7634.544} C_VEL
LIN {X 0,Y 468.585,Z 530.067,A -85,B 0,C 180,E1 -7634.908,E2 -7634.908} C_VEL
LIN {X 0,Y 469.732,Z 541.897,A -85,B 0,C 180,E1 -7635.375,E2 -7635.375} C_VEL
LIN {X 0,Y 469.276,Z 552.975,A -85,B 0,C 180,E1 -7635.915,E2 -7635.915} C_VEL
LIN {X 0,Y 468.765,Z 564.933,A -85,B 0,C 180,E1 -7636.673,E2 -7636.673} C_VEL
LIN {X 0,Y 468.256,Z 576.024,A -85,B 0,C 180,E1 -7637.571,E2 -7637.571} C_VEL
LIN {X 0,Y 467.849,Z 585.554,A -85,B 0,C 180,E1 -7638.519,E2 -7638.519} C_VEL
LIN {X 0,Y 467.487,Z 594.571,A -85,B 0,C 180,E1 -7639.607,E2 -7639.607} C_VEL
LIN {X 0,Y 467.22,Z 603.406,A -85,B 0,C 180,E1 -7640.912,E2 -7640.912} C_VEL
LIN {X 0,Y 467.043,Z 610.485,A -85,B 0,C 180,E1 -7642.216,E2 -7642.216} C_VEL
LIN {X 0,Y 466.973,Z 616.702,A -85,B 0,C 180,E1 -7643.655,E2 -7643.655} C_VEL
LIN {X 0,Y 466.958,Z 621.923,A -85,B 0,C 180,E1 -7645.252,E2 -7645.252} C_VEL
LIN {X 0,Y 466.968,Z 624.955,A -85,B 0,C 180,E1 -7646.548,E2 -7646.548} C_VEL
LIN {X 0,Y 466.957,Z 626.4,A -85,B 0,C 180,E1 -7647.412,E2 -7647.412} C_VEL
LIN {X 0,Y 467.037,Z 628.075,A -85,B 0,C 180,E1 -7649.138,E2 -7649.138} C_VEL
LIN {X 0,Y 467.023,Z 628.3,A -85,B 0,C 180,E1 -7650,E2 -7650} C_VEL
LIN {X 0,Y 467.037,Z 628.082,A -85,B 0,C 180,E1 -7650.862,E2 -7650.862} C_VEL
LIN {X 0,Y 466.954,Z 626.423,A -85,B 0,C 180,E1 -7652.588,E2 -7652.588} C_VEL
LIN {X 0,Y 466.965,Z 624.986,A -85,B 0,C 180,E1 -7653.451,E2 -7653.451} C_VEL
LIN {X 0,Y 466.957,Z 621.961,A -85,B 0,C 180,E1 -7654.748,E2 -7654.748} C_VEL
LIN {X 0,Y 466.961,Z 616.797,A -85,B 0,C 180,E1 -7656.332,E2 -7656.332} C_VEL
LIN {X 0,Y 467.042,Z 610.545,A -85,B 0,C 180,E1 -7657.783,E2 -7657.783} C_VEL
LIN {X 0,Y 467.22,Z 603.471,A -85,B 0,C 180,E1 -7659.087,E2 -7659.087} C_VEL
LIN {X 0,Y 467.486,Z 594.635,A -85,B 0,C 180,E1 -7660.393,E2 -7660.393} C_VEL
LIN {X 0,Y 467.934,Z 584.616,A -85,B 0,C 180,E1 -7661.588,E2 -7661.588} C_VEL
LIN {X 0,Y 468.306,Z 574.517,A -85,B 0,C 180,E1 -7662.568,E2 -7662.568} C_VEL
LIN {X 0,Y 468.847,Z 563.353,A -85,B 0,C 180,E1 -7663.435,E2 -7663.435} C_VEL
LIN {X 0,Y 469.339,Z 550.861,A -85,B 0,C 180,E1 -7664.194,E2 -7664.194} C_VEL
LIN {X 0,Y 469.656,Z 540.354,A -85,B 0,C 180,E1 -7664.682,E2 -7664.682} C_VEL
LIN {X 0,Y 468.523,Z 530.007,A -85,B 0,C 180,E1 -7665.08,E2 -7665.08} C_VEL
LIN {X 0,Y 467.289,Z 516.378,A -85,B 0,C 180,E1 -7665.455,E2 -7665.455} C_VEL
LIN {X 0,Y 467.556,Z 503.293,A -85,B 0,C 180,E1 -7668.4,E2 -7668.4} C_VEL
LIN {X 0,Y 467.891,Z 488.87,A -85,B 0,C 180,E1 -7671.654,E2 -7671.654} C_VEL
LIN {X 0,Y 468.285,Z 473.761,A -85,B 0,C 180,E1 -7675.086,E2 -7675.086} C_VEL
LIN {X 0,Y 468.71,Z 459.285,A -85,B 0,C 180,E1 -7678.429,E2 -7678.429} C_VEL
LIN {X 0,Y 469.173,Z 445.796,A -85,B 0,C 180,E1 -7681.62,E2 -7681.62} C_VEL
LIN {X 0,Y 469.668,Z 433.375,A -85,B 0,C 180,E1 -7684.654,E2 -7684.654} C_VEL
LIN {X 0,Y 470.013,Z 426.455,A -85,B 0,C 180,E1 -7686.396,E2 -7686.396} C_VEL
LIN {X 0,Y 468.508,Z 417.938,A -85,B 0,C 180,E1 -7688.735,E2 -7688.735} C_VEL
LIN {X 0,Y 467.638,Z 413.237,A -85,B 0,C 180,E1 -7690.121,E2 -7690.121} C_VEL
LIN {X 0,Y 467.587,Z 413.243,A -85,B 0,C 180,E1 -7692.567,E2 -7692.567} C_VEL
LIN {X 0,Y 467.572,Z 413.247,A -85,B 0,C 180,E1 -7695.053,E2 -7695.053} C_VEL
LIN {X 0,Y 467.59,Z 413.24,A -85,B 0,C 180,E1 -7697.44,E2 -7697.44} C_VEL
LIN {X 0,Y 467.584,Z 413.242,A -85,B 0,C 180,E1 -7700.855,E2 -7700.855} C_VEL
LIN {X 0,Y 467.563,Z 413.246,A -85,B 0,C 180,E1 -7704.26,E2 -7704.26} C_VEL
LIN {X 0,Y 467.583,Z 413.24,A -85,B 0,C 180,E1 -7707.321,E2 -7707.321} C_VEL
LIN {X 0,Y 467.571,Z 413.245,A -85,B 0,C 180,E1 -7710.667,E2 -7710.667} C_VEL
LIN {X 0,Y 467.629,Z 413.235,A -85,B 0,C 180,E1 -7713.2,E2 -7713.2} C_VEL
LIN {X 0,Y 467.594,Z 413.241,A -85,B 0,C 180,E1 -7716.468,E2 -7716.468} C_VEL
LIN {X 0,Y 467.626,Z 413.238,A -85,B 0,C 180,E1 -7719.777,E2 -7719.777} C_VEL
LIN {X 0,Y 467.611,Z 413.24,A -85,B 0,C 180,E1 -7722.507,E2 -7722.507} C_VEL
LIN {X 0,Y 467.608,Z 413.238,A -85,B 0,C 180,E1 -7725.197,E2 -7725.197} C_VEL
LIN {X 0,Y 467.685,Z 413.23,A -85,B 0,C 180,E1 -7727.855,E2 -7727.855} C_VEL
LIN {X 0,Y 467.672,Z 413.23,A -85,B 0,C 180,E1 -7731.357,E2 -7731.357} C_VEL
LIN {X 0,Y 467.745,Z 413.224,A -85,B 0,C 180,E1 -7733.963,E2 -7733.963} C_VEL
LIN {X 0,Y 467.864,Z 413.207,A -85,B 0,C 180,E1 -7737.417,E2 -7737.417} C_VEL
LIN {X 0,Y 467.885,Z 413.206,A -85,B 0,C 180,E1 -7740,E2 -7740} C_VEL
LIN {X 0,Y 467.861,Z 413.207,A -85,B 0,C 180,E1 -7742.583,E2 -7742.583} C_VEL
LIN {X 0,Y 467.745,Z 413.223,A -85,B 0,C 180,E1 -7746.038,E2 -7746.038} C_VEL
LIN {X 0,Y 467.684,Z 413.229,A -85,B 0,C 180,E1 -7748.643,E2 -7748.643} C_VEL
LIN {X 0,Y 467.658,Z 413.234,A -85,B 0,C 180,E1 -7752.146,E2 -7752.146} C_VEL
LIN {X 0,Y 467.641,Z 413.236,A -85,B 0,C 180,E1 -7755.695,E2 -7755.695} C_VEL
LIN {X 0,Y 467.62,Z 413.236,A -85,B 0,C 180,E1 -7758.765,E2 -7758.765} C_VEL
LIN {X 0,Y 467.584,Z 413.242,A -85,B 0,C 180,E1 -7761.269,E2 -7761.269} C_VEL
LIN {X 0,Y 467.576,Z 413.245,A -85,B 0,C 180,E1 -7763.943,E2 -7763.943} C_VEL
LIN {X 0,Y 467.619,Z 413.236,A -85,B 0,C 180,E1 -7766.8,E2 -7766.8} C_VEL
LIN {X 0,Y 467.556,Z 413.247,A -85,B 0,C 180,E1 -7769.738,E2 -7769.738} C_VEL
LIN {X 0,Y 467.586,Z 413.241,A -85,B 0,C 180,E1 -7772.759,E2 -7772.759} C_VEL
LIN {X 0,Y 467.559,Z 413.247,A -85,B 0,C 180,E1 -7775.89,E2 -7775.89} C_VEL
LIN {X 0,Y 467.585,Z 413.241,A -85,B 0,C 180,E1 -7779.145,E2 -7779.145} C_VEL
LIN {X 0,Y 467.589,Z 413.24,A -85,B 0,C 180,E1 -7782.567,E2 -7782.567} C_VEL
LIN {X 0,Y 467.574,Z 413.242,A -85,B 0,C 180,E1 -7785.054,E2 -7785.054} C_VEL
LIN {X 0,Y 467.591,Z 413.241,A -85,B 0,C 180,E1 -7787.44,E2 -7787.44} C_VEL
LIN {X 0,Y 467.585,Z 413.24,A -85,B 0,C 180,E1 -7790.856,E2 -7790.856} C_VEL
LIN {X 0,Y 467.566,Z 413.245,A -85,B 0,C 180,E1 -7794.261,E2 -7794.261} C_VEL
LIN {X 0,Y 467.586,Z 413.242,A -85,B 0,C 180,E1 -7797.321,E2 -7797.321} C_VEL
LIN {X 0,Y 467.581,Z 413.241,A -85,B 0,C 180,E1 -7800.666,E2 -7800.666} C_VEL
LIN {X 0,Y 467.62,Z 413.238,A -85,B 0,C 180,E1 -7803.2,E2 -7803.2} C_VEL
LIN {X 0,Y 467.596,Z 413.239,A -85,B 0,C 180,E1 -7806.468,E2 -7806.468} C_VEL
LIN {X 0,Y 467.629,Z 413.238,A -85,B 0,C 180,E1 -7809.778,E2 -7809.778} C_VEL
LIN {X 0,Y 467.613,Z 413.237,A -85,B 0,C 180,E1 -7812.507,E2 -7812.507} C_VEL
LIN {X 0,Y 467.601,Z 413.24,A -85,B 0,C 180,E1 -7815.425,E2 -7815.425} C_VEL
LIN {X 0,Y 466.921,Z 413.327,A -85,B 0,C 180,E1 -7815.905,E2 -7815.905} C_VEL
LIN {X 0,Y 464.088,Z 413.678,A -85,B 0,C 180,E1 -7816.657,E2 -7816.657} C_VEL
LIN {X 0,Y 461.269,Z 414.029,A -85,B 0,C 180,E1 -7817.417,E2 -7817.417} C_VEL
LIN {X 0,Y 460.627,Z 414.107,A -85,B 0,C 180,E1 -7817.907,E2 -7817.907} C_VEL
LIN {X 0,Y 460.647,Z 414.113,A -85,B 0,C 180,E1 -7818.254,E2 -7818.254} C_VEL
LIN {X 0,Y 463.498,Z 425.094,A -85,B 0,C 180,E1 -7818.964,E2 -7818.964} C_VEL
LIN {X 0,Y 463.155,Z 436.116,A -85,B 0,C 180,E1 -7819.73,E2 -7819.73} C_VEL
LIN {X 0,Y 462.595,Z 447.354,A -85,B 0,C 180,E1 -7820.711,E2 -7820.711} C_VEL
LIN {X 0,Y 462.142,Z 456.78,A -85,B 0,C 180,E1 -7821.744,E2 -7821.744} C_VEL
LIN {X 0,Y 461.633,Z 466.053,A -85,B 0,C 180,E1 -7823.005,E2 -7823.005} C_VEL
LIN {X 0,Y 461.292,Z 473.813,A -85,B 0,C 180,E1 -7824.317,E2 -7824.317} C_VEL
LIN {X 0,Y 460.939,Z 480.04,A -85,B 0,C 180,E1 -7825.628,E2 -7825.628} C_VEL
LIN {X 0,Y 460.63,Z 484.987,A -85,B 0,C 180,E1 -7826.939,E2 -7826.939} C_VEL
LIN {X 0,Y 460.453,Z 488.82,A -85,B 0,C 180,E1 -7828.251,E2 -7828.251} C_VEL
LIN {X 0,Y 460.273,Z 492.365,A -85,B 0,C 180,E1 -7830,E2 -7830} C_VEL
LIN {X 0,Y 460.133,Z 493.563,A -85,B 0,C 180,E1 -7830.875,E2 -7830.875} C_VEL
LIN {X 0,Y 460.198,Z 494.32,A -85,B 0,C 180,E1 -7831.75,E2 -7831.75} C_VEL
LIN {X 0,Y 460.156,Z 494.704,A -85,B 0,C 180,E1 -7833.503,E2 -7833.503} C_VEL
LIN {X 0,Y 460.203,Z 494.335,A -85,B 0,C 180,E1 -7834.379,E2 -7834.379} C_VEL
LIN {X 0,Y 460.311,Z 493.557,A -85,B 0,C 180,E1 -7835.256,E2 -7835.256} C_VEL
LIN {X 0,Y 460.427,Z 490.808,A -85,B 0,C 180,E1 -7837.014,E2 -7837.014} C_VEL
LIN {X 0,Y 460.577,Z 487.64,A -85,B 0,C 180,E1 -7838.335,E2 -7838.335} C_VEL
LIN {X 0,Y 460.845,Z 483.411,A -85,B 0,C 180,E1 -7839.657,E2 -7839.657} C_VEL
LIN {X 0,Y 461.159,Z 478.003,A -85,B 0,C 180,E1 -7840.982,E2 -7840.982} C_VEL
LIN {X 0,Y 461.416,Z 471.242,A -85,B 0,C 180,E1 -7842.312,E2 -7842.312} C_VEL
LIN {X 0,Y 461.958,Z 462.691,A -85,B 0,C 180,E1 -7843.64,E2 -7843.64} C_VEL
LIN {X 0,Y 462.4,Z 453.906,A -85,B 0,C 180,E1 -7844.749,E2 -7844.749} C_VEL
LIN {X 0,Y 462.855,Z 444.207,A -85,B 0,C 180,E1 -7845.749,E2 -7845.749} C_VEL
LIN {X 0,Y 463.318,Z 433.45,A -85,B 0,C 180,E1 -7846.638,E2 -7846.638} C_VEL
LIN {X 0,Y 463.597,Z 424.456,A -85,B 0,C 180,E1 -7847.24,E2 -7847.24} C_VEL
LIN {X 0,Y 460.575,Z 414.116,A -85,B 0,C 180,E1 -7847.942,E2 -7847.942} C_VEL
LIN {X 0,Y 460.556,Z 414.118,A -85,B 0,C 180,E1 -7850.547,E2 -7850.547} C_VEL
LIN {X 0,Y 460.536,Z 414.115,A -85,B 0,C 180,E1 -7853.704,E2 -7853.704} C_VEL
LIN {X 0,Y 460.561,Z 414.119,A -85,B 0,C 180,E1 -7856.266,E2 -7856.266} C_VEL
LIN {X 0,Y 460.544,Z 414.113,A -85,B 0,C 180,E1 -7859.231,E2 -7859.231} C_VEL
LIN {X 0,Y 460.536,Z 414.121,A -85,B 0,C 180,E1 -7862.284,E2 -7862.284} C_VEL
LIN {X 0,Y 460.518,Z 414.117,A -85,B 0,C 180,E1 -7865.445,E2 -7865.445} C_VEL
LIN {X 0,Y 460.549,Z 414.113,A -85,B 0,C 180,E1 -7868.898,E2 -7868.898} C_VEL
LIN {X 0,Y 460.527,Z 414.122,A -85,B 0,C 180,E1 -7872.181,E2 -7872.181} C_VEL
LIN {X 0,Y 460.522,Z 414.117,A -85,B 0,C 180,E1 -7875.412,E2 -7875.412} C_VEL
LIN {X 0,Y 460.537,Z 414.117,A -85,B 0,C 180,E1 -7878.397,E2 -7878.397} C_VEL
LIN {X 0,Y 460.53,Z 414.115,A -85,B 0,C 180,E1 -7881.267,E2 -7881.267} C_VEL
LIN {X 0,Y 460.515,Z 414.118,A -85,B 0,C 180,E1 -7884.554,E2 -7884.554} C_VEL
LIN {X 0,Y 460.536,Z 414.119,A -85,B 0,C 180,E1 -7887.716,E2 -7887.716} C_VEL
LIN {X 0,Y 460.544,Z 414.113,A -85,B 0,C 180,E1 -7890.769,E2 -7890.769} C_VEL
LIN {X 0,Y 460.56,Z 414.118,A -85,B 0,C 180,E1 -7893.734,E2 -7893.734} C_VEL
LIN {X 0,Y 460.549,Z 414.113,A -85,B 0,C 180,E1 -7896.624,E2 -7896.624} C_VEL
LIN {X 0,Y 460.556,Z 414.116,A -85,B 0,C 180,E1 -7899.453,E2 -7899.453} C_VEL
LIN {X 0,Y 460.554,Z 414.114,A -85,B 0,C 180,E1 -7902.23,E2 -7902.23} C_VEL
LIN {X 0,Y 460.57,Z 414.11,A -85,B 0,C 180,E1 -7904.965,E2 -7904.965} C_VEL
LIN {X 0,Y 460.614,Z 414.265,A -85,B 0,C 180,E1 -7906.491,E2 -7906.491} C_VEL
LIN {X 0,Y 463.023,Z 423.062,A -85,B 0,C 180,E1 -7907.072,E2 -7907.072} C_VEL
LIN {X 0,Y 462.631,Z 434.216,A -85,B 0,C 180,E1 -7907.832,E2 -7907.832} C_VEL
LIN {X 0,Y 462.185,Z 445.621,A -85,B 0,C 180,E1 -7908.821,E2 -7908.821} C_VEL
LIN {X 0,Y 461.871,Z 455.831,A -85,B 0,C 180,E1 -7909.922,E2 -7909.922} C_VEL
LIN {X 0,Y 461.416,Z 464.182,A -85,B 0,C 180,E1 -7911.018,E2 -7911.018} C_VEL
LIN {X 0,Y 461.03,Z 472.378,A -85,B 0,C 180,E1 -7912.345,E2 -7912.345} C_VEL
LIN {X 0,Y 460.798,Z 477.884,A -85,B 0,C 180,E1 -7913.431,E2 -7913.431} C_VEL
LIN {X 0,Y 460.481,Z 483.338,A -85,B 0,C 180,E1 -7914.746,E2 -7914.746} C_VEL
LIN {X 0,Y 460.463,Z 487.583,A -85,B 0,C 180,E1 -7916.061,E2 -7916.061} C_VEL
LIN {X 0,Y 460.172,Z 490.814,A -85,B 0,C 180,E1 -7917.374,E2 -7917.374} C_VEL
LIN {X 0,Y 460.21,Z 492.416,A -85,B 0,C 180,E1 -7918.25,E2 -7918.25} C_VEL
LIN {X 0,Y 460.131,Z 493.587,A -85,B 0,C 180,E1 -7919.125,E2 -7919.125} C_VEL
LIN {X 0,Y 460.128,Z 494.732,A -85,B 0,C 180,E1 -7920.875,E2 -7920.875} C_VEL
LIN {X 0,Y 460.201,Z 494.709,A -85,B 0,C 180,E1 -7921.75,E2 -7921.75} C_VEL
LIN {X 0,Y 460.234,Z 493.442,A -85,B 0,C 180,E1 -7923.502,E2 -7923.502} C_VEL
LIN {X 0,Y 460.314,Z 492.226,A -85,B 0,C 180,E1 -7924.378,E2 -7924.378} C_VEL
LIN {X 0,Y 460.51,Z 489.563,A -85,B 0,C 180,E1 -7925.693,E2 -7925.693} C_VEL
LIN {X 0,Y 460.733,Z 485.879,A -85,B 0,C 180,E1 -7927.009,E2 -7927.009} C_VEL
LIN {X 0,Y 460.95,Z 481.052,A -85,B 0,C 180,E1 -7928.328,E2 -7928.328} C_VEL
LIN {X 0,Y 461.305,Z 474.898,A -85,B 0,C 180,E1 -7929.647,E2 -7929.647} C_VEL
LIN {X 0,Y 461.667,Z 467.228,A -85,B 0,C 180,E1 -7930.97,E2 -7930.97} C_VEL
LIN {X 0,Y 462.083,Z 459.35,A -85,B 0,C 180,E1 -7932.071,E2 -7932.071} C_VEL
LIN {X 0,Y 462.458,Z 449.641,A -85,B 0,C 180,E1 -7933.177,E2 -7933.177} C_VEL
LIN {X 0,Y 463.04,Z 438.782,A -85,B 0,C 180,E1 -7934.167,E2 -7934.167} C_VEL
LIN {X 0,Y 463.459,Z 428.239,A -85,B 0,C 180,E1 -7934.939,E2 -7934.939} C_VEL
LIN {X 0,Y 463.516,Z 424.703,A -85,B 0,C 180,E1 -7935.162,E2 -7935.162} C_VEL
LIN {X 0,Y 460.625,Z 414.111,A -85,B 0,C 180,E1 -7935.885,E2 -7935.885} C_VEL
LIN {X 0,Y 460.573,Z 414.12,A -85,B 0,C 180,E1 -7939.615,E2 -7939.615} C_VEL
LIN {X 0,Y 460.514,Z 414.125,A -85,B 0,C 180,E1 -7942.428,E2 -7942.428} C_VEL
LIN {X 0,Y 460.556,Z 414.118,A -85,B 0,C 180,E1 -7945.798,E2 -7945.798} C_VEL
LIN {X 0,Y 460.559,Z 414.115,A -85,B 0,C 180,E1 -7948.233,E2 -7948.233} C_VEL
LIN {X 0,Y 460.524,Z 414.122,A -85,B 0,C 180,E1 -7951.283,E2 -7951.283} C_VEL
LIN {X 0,Y 460.535,Z 414.12,A -85,B 0,C 180,E1 -7954.505,E2 -7954.505} C_VEL
LIN {X 0,Y 460.504,Z 414.122,A -85,B 0,C 180,E1 -7957.623,E2 -7957.623} C_VEL
LIN {X 0,Y 460.546,Z 414.118,A -85,B 0,C 180,E1 -7960.269,E2 -7960.269} C_VEL
LIN {X 0,Y 460.503,Z 414.124,A -85,B 0,C 180,E1 -7963.375,E2 -7963.375} C_VEL
LIN {X 0,Y 460.503,Z 414.124,A -85,B 0,C 180,E1 -7966.625,E2 -7966.625} C_VEL
LIN {X 0,Y 460.577,Z 414.26,A -85,B 0,C 180,E1 -7969.237,E2 -7969.237} C_VEL
LIN {X 0,Y 462.565,Z 424.217,A -85,B 0,C 180,E1 -7972.192,E2 -7972.192} C_VEL
LIN {X 0,Y 463.306,Z 428.892,A -85,B 0,C 180,E1 -7973.511,E2 -7973.511} C_VEL
LIN {X 0,Y 462.514,Z 441.719,A -85,B 0,C 180,E1 -7976.836,E2 -7976.836} C_VEL
LIN {X 0,Y 462.069,Z 452.895,A -85,B 0,C 180,E1 -7979.62,E2 -7979.62} C_VEL
LIN {X 0,Y 461.559,Z 466.12,A -85,B 0,C 180,E1 -7982.819,E2 -7982.819} C_VEL
LIN {X 0,Y 461.159,Z 478.3,A -85,B 0,C 180,E1 -7985.702,E2 -7985.702} C_VEL
LIN {X 0,Y 460.717,Z 492.425,A -85,B 0,C 180,E1 -7988.993,E2 -7988.993} C_VEL
LIN {X 0,Y 460.419,Z 506.382,A -85,B 0,C 180,E1 -7992.224,E2 -7992.224} C_VEL
LIN {X 0,Y 460.213,Z 515.276,A -85,B 0,C 180,E1 -7994.28,E2 -7994.28} C_VEL
LIN {X 0,Y 461.653,Z 529.951,A -85,B 0,C 180,E1 -7994.694,E2 -7994.694} C_VEL
LIN {X 0,Y 462.534,Z 539.738,A -85,B 0,C 180,E1 -7995.086,E2 -7995.086} C_VEL
LIN {X 0,Y 462.674,Z 544.699,A -85,B 0,C 180,E1 -7995.316,E2 -7995.316} C_VEL
LIN {X 0,Y 462.068,Z 557.571,A -85,B 0,C 180,E1 -7996.027,E2 -7996.027} C_VEL
LIN {X 0,Y 461.57,Z 568.321,A -85,B 0,C 180,E1 -7996.797,E2 -7996.797} C_VEL
LIN {X 0,Y 461.143,Z 579.366,A -85,B 0,C 180,E1 -7997.792,E2 -7997.792} C_VEL
LIN {X 0,Y 460.675,Z 588.39,A -85,B 0,C 180,E1 -7998.784,E2 -7998.784} C_VEL
LIN {X 0,Y 460.277,Z 598.241,A -85,B 0,C 180,E1 -8000.109,E2 -8000.109} C_VEL
LIN {X 0,Y 460.042,Z 606.12,A -85,B 0,C 180,E1 -8001.434,E2 -8001.434} C_VEL
LIN {X 0,Y 459.927,Z 613.411,A -85,B 0,C 180,E1 -8002.978,E2 -8002.978} C_VEL
LIN {X 0,Y 459.911,Z 618.282,A -85,B 0,C 180,E1 -8004.299,E2 -8004.299} C_VEL
LIN {X 0,Y 459.921,Z 622.013,A -85,B 0,C 180,E1 -8005.618,E2 -8005.618} C_VEL
LIN {X 0,Y 459.924,Z 623.938,A -85,B 0,C 180,E1 -8006.496,E2 -8006.496} C_VEL
LIN {X 0,Y 459.916,Z 625.384,A -85,B 0,C 180,E1 -8007.372,E2 -8007.372} C_VEL
LIN {X 0,Y 460.021,Z 627.064,A -85,B 0,C 180,E1 -8009.124,E2 -8009.124} C_VEL
LIN {X 0,Y 460.008,Z 627.289,A -85,B 0,C 180,E1 -8010,E2 -8010} C_VEL
LIN {X 0,Y 460.021,Z 627.072,A -85,B 0,C 180,E1 -8010.875,E2 -8010.875} C_VEL
LIN {X 0,Y 459.913,Z 625.409,A -85,B 0,C 180,E1 -8012.627,E2 -8012.627} C_VEL
LIN {X 0,Y 459.921,Z 623.97,A -85,B 0,C 180,E1 -8013.504,E2 -8013.504} C_VEL
LIN {X 0,Y 459.911,Z 620.942,A -85,B 0,C 180,E1 -8014.821,E2 -8014.821} C_VEL
LIN {X 0,Y 459.934,Z 616.847,A -85,B 0,C 180,E1 -8016.14,E2 -8016.14} C_VEL
LIN {X 0,Y 459.972,Z 610.547,A -85,B 0,C 180,E1 -8017.683,E2 -8017.683} C_VEL
LIN {X 0,Y 460.103,Z 603.684,A -85,B 0,C 180,E1 -8019.008,E2 -8019.008} C_VEL
LIN {X 0,Y 460.368,Z 595.195,A -85,B 0,C 180,E1 -8020.333,E2 -8020.333} C_VEL
LIN {X 0,Y 460.731,Z 586.508,A -85,B 0,C 180,E1 -8021.438,E2 -8021.438} C_VEL
LIN {X 0,Y 461.246,Z 576.439,A -85,B 0,C 180,E1 -8022.482,E2 -8022.482} C_VEL
LIN {X 0,Y 461.652,Z 566.688,A -85,B 0,C 180,E1 -8023.312,E2 -8023.312} C_VEL
LIN {X 0,Y 462.148,Z 555.464,A -85,B 0,C 180,E1 -8024.082,E2 -8024.082} C_VEL
LIN {X 0,Y 462.708,Z 543.036,A -85,B 0,C 180,E1 -8024.739,E2 -8024.739} C_VEL
LIN {X 0,Y 461.593,Z 530.459,A -85,B 0,C 180,E1 -8025.256,E2 -8025.256} C_VEL
LIN {X 0,Y 460.335,Z 517.085,A -85,B 0,C 180,E1 -8025.629,E2 -8025.629} C_VEL
LIN {X 0,Y 460.207,Z 515.494,A -85,B 0,C 180,E1 -8025.663,E2 -8025.663} C_VEL
LIN {X 0,Y 460.47,Z 502.29,A -85,B 0,C 180,E1 -8028.694,E2 -8028.694} C_VEL
LIN {X 0,Y 460.837,Z 488.171,A -85,B 0,C 180,E1 -8031.94,E2 -8031.94} C_VEL
LIN {X 0,Y 461.229,Z 473.847,A -85,B 0,C 180,E1 -8035.255,E2 -8035.255} C_VEL
LIN {X 0,Y 461.729,Z 459.416,A -85,B 0,C 180,E1 -8038.65,E2 -8038.65} C_VEL
LIN {X 0,Y 462.201,Z 446.207,A -85,B 0,C 180,E1 -8041.836,E2 -8041.836} C_VEL
LIN {X 0,Y 462.738,Z 433.897,A -85,B 0,C 180,E1 -8044.9,E2 -8044.9} C_VEL
LIN {X 0,Y 463.064,Z 427.852,A -85,B 0,C 180,E1 -8046.448,E2 -8046.448} C_VEL
LIN {X 0,Y 461.725,Z 420.064,A -85,B 0,C 180,E1 -8048.614,E2 -8048.614} C_VEL
LIN {X 0,Y 460.584,Z 414.116,A -85,B 0,C 180,E1 -8050.403,E2 -8050.403} C_VEL
LIN {X 0,Y 460.501,Z 414.127,A -85,B 0,C 180,E1 -8053.375,E2 -8053.375} C_VEL
LIN {X 0,Y 460.51,Z 414.125,A -85,B 0,C 180,E1 -8056.626,E2 -8056.626} C_VEL
LIN {X 0,Y 460.544,Z 414.118,A -85,B 0,C 180,E1 -8059.73,E2 -8059.73} C_VEL
LIN {X 0,Y 460.528,Z 414.122,A -85,B 0,C 180,E1 -8062.519,E2 -8062.519} C_VEL
LIN {X 0,Y 460.549,Z 414.118,A -85,B 0,C 180,E1 -8065.624,E2 -8065.624} C_VEL
LIN {X 0,Y 460.538,Z 414.119,A -85,B 0,C 180,E1 -8068.745,E2 -8068.745} C_VEL
LIN {X 0,Y 460.59,Z 414.115,A -85,B 0,C 180,E1 -8072.252,E2 -8072.252} C_VEL
LIN {X 0,Y 460.561,Z 414.117,A -85,B 0,C 180,E1 -8074.706,E2 -8074.706} C_VEL
LIN {X 0,Y 460.514,Z 414.122,A -85,B 0,C 180,E1 -8077.572,E2 -8077.572} C_VEL
LIN {X 0,Y 460.571,Z 414.117,A -85,B 0,C 180,E1 -8080.385,E2 -8080.385} C_VEL
LIN {X 0,Y 460.567,Z 414.114,A -85,B 0,C 180,E1 -8083.146,E2 -8083.146} C_VEL
LIN {X 0,Y 460.557,Z 414.118,A -85,B 0,C 180,E1 -8085.868,E2 -8085.868} C_VEL
LIN {X 0,Y 460.632,Z 414.108,A -85,B 0,C 180,E1 -8088.56,E2 -8088.56} C_VEL
LIN {X 0,Y 460.622,Z 414.107,A -85,B 0,C 180,E1 -8091.224,E2 -8091.224} C_VEL
LIN {X 0,Y 460.709,Z 414.1,A -85,B 0,C 180,E1 -8093.87,E2 -8093.87} C_VEL
LIN {X 0,Y 460.828,Z 414.083,A -85,B 0,C 180,E1 -8097.378,E2 -8097.378} C_VEL
LIN {X 0,Y 460.855,Z 414.082,A -85,B 0,C 180,E1 -8100,E2 -8100} C_VEL
LIN {X 0,Y 460.801,Z 414.086,A -85,B 0,C 180,E1 -8102.623,E2 -8102.623} C_VEL
LIN {X 0,Y 460.712,Z 414.099,A -85,B 0,C 180,E1 -8106.13,E2 -8106.13} C_VEL
LIN {X 0,Y 460.631,Z 414.107,A -85,B 0,C 180,E1 -8108.776,E2 -8108.776} C_VEL
LIN {X 0,Y 460.615,Z 414.11,A -85,B 0,C 180,E1 -8112.445,E2 -8112.445} C_VEL
LIN {X 0,Y 460.602,Z 414.113,A -85,B 0,C 180,E1 -8115.998,E2 -8115.998} C_VEL
LIN {X 0,Y 460.573,Z 414.113,A -85,B 0,C 180,E1 -8118.902,E2 -8118.902} C_VEL
LIN {X 0,Y 460.518,Z 414.122,A -85,B 0,C 180,E1 -8121.486,E2 -8121.486} C_VEL
LIN {X 0,Y 460.545,Z 414.119,A -85,B 0,C 180,E1 -8124.332,E2 -8124.332} C_VEL
LIN {X 0,Y 460.581,Z 414.113,A -85,B 0,C 180,E1 -8127.244,E2 -8127.244} C_VEL
LIN {X 0,Y 460.513,Z 414.124,A -85,B 0,C 180,E1 -8130.24,E2 -8130.24} C_VEL
LIN {X 0,Y 460.532,Z 414.12,A -85,B 0,C 180,E1 -8133.325,E2 -8133.325} C_VEL
LIN {X 0,Y 460.481,Z 414.126,A -85,B 0,C 180,E1 -8136.529,E2 -8136.529} C_VEL
LIN {X 0,Y 460.547,Z 414.117,A -85,B 0,C 180,E1 -8138.898,E2 -8138.898} C_VEL
LIN {X 0,Y 460.526,Z 414.123,A -85,B 0,C 180,E1 -8142.181,E2 -8142.181} C_VEL
LIN {X 0,Y 460.523,Z 414.122,A -85,B 0,C 180,E1 -8145.412,E2 -8145.412} C_VEL
LIN {X 0,Y 460.538,Z 414.119,A -85,B 0,C 180,E1 -8148.397,E2 -8148.397} C_VEL
LIN {X 0,Y 460.53,Z 414.121,A -85,B 0,C 180,E1 -8151.267,E2 -8151.267} C_VEL
LIN {X 0,Y 460.516,Z 414.121,A -85,B 0,C 180,E1 -8154.555,E2 -8154.555} C_VEL
LIN {X 0,Y 460.536,Z 414.122,A -85,B 0,C 180,E1 -8157.716,E2 -8157.716} C_VEL
LIN {X 0,Y 460.551,Z 414.117,A -85,B 0,C 180,E1 -8160.77,E2 -8160.77} C_VEL
LIN {X 0,Y 460.567,Z 414.117,A -85,B 0,C 180,E1 -8163.735,E2 -8163.735} C_VEL
LIN {X 0,Y 460.55,Z 414.116,A -85,B 0,C 180,E1 -8166.624,E2 -8166.624} C_VEL
LIN {X 0,Y 460.557,Z 414.118,A -85,B 0,C 180,E1 -8169.453,E2 -8169.453} C_VEL
LIN {X 0,Y 460.564,Z 414.116,A -85,B 0,C 180,E1 -8172.23,E2 -8172.23} C_VEL
LIN {X 0,Y 460.57,Z 414.117,A -85,B 0,C 180,E1 -8174.965,E2 -8174.965} C_VEL
LIN {X 0,Y 460.627,Z 414.107,A -85,B 0,C 180,E1 -8177.907,E2 -8177.907} C_VEL
LIN {X 0,Y 460.611,Z 414.955,A -85,B 0,C 180,E1 -8178.171,E2 -8178.171} C_VEL
LIN {X 0,Y 460.504,Z 417.553,A -85,B 0,C 180,E1 -8178.421,E2 -8178.421} C_VEL
LIN {X 0,Y 460.065,Z 423.057,A -85,B 0,C 180,E1 -8178.709,E2 -8178.709} C_VEL
LIN {X 0,Y 457.011,Z 436.302,A -85,B 0,C 180,E1 -8179.467,E2 -8179.467} C_VEL
LIN {X 0,Y 456.063,Z 441.369,A -85,B 0,C 180,E1 -8179.887,E2 -8179.887} C_VEL
LIN {X 0,Y 455.57,Z 452.43,A -85,B 0,C 180,E1 -8180.964,E2 -8180.964} C_VEL
LIN {X 0,Y 455.055,Z 461.135,A -85,B 0,C 180,E1 -8182.01,E2 -8182.01} C_VEL
LIN {X 0,Y 454.712,Z 468.707,A -85,B 0,C 180,E1 -8183.121,E2 -8183.121} C_VEL
LIN {X 0,Y 454.233,Z 476.121,A -85,B 0,C 180,E1 -8184.451,E2 -8184.451} C_VEL
LIN {X 0,Y 453.883,Z 482.943,A -85,B 0,C 180,E1 -8186.005,E2 -8186.005} C_VEL
LIN {X 0,Y 453.611,Z 487.479,A -85,B 0,C 180,E1 -8187.336,E2 -8187.336} C_VEL
LIN {X 0,Y 453.449,Z 489.912,A -85,B 0,C 180,E1 -8188.224,E2 -8188.224} C_VEL
LIN {X 0,Y 453.26,Z 493.431,A -85,B 0,C 180,E1 -8190,E2 -8190} C_VEL
LIN {X 0,Y 453.112,Z 494.617,A -85,B 0,C 180,E1 -8190.889,E2 -8190.889} C_VEL
LIN {X 0,Y 453.18,Z 495.349,A -85,B 0,C 180,E1 -8191.778,E2 -8191.778} C_VEL
LIN {X 0,Y 453.131,Z 495.71,A -85,B 0,C 180,E1 -8193.557,E2 -8193.557} C_VEL
LIN {X 0,Y 453.185,Z 495.329,A -85,B 0,C 180,E1 -8194.447,E2 -8194.447} C_VEL
LIN {X 0,Y 453.307,Z 494.525,A -85,B 0,C 180,E1 -8195.338,E2 -8195.338} C_VEL
LIN {X 0,Y 453.424,Z 491.753,A -85,B 0,C 180,E1 -8197.123,E2 -8197.123} C_VEL
LIN {X 0,Y 453.594,Z 488.559,A -85,B 0,C 180,E1 -8198.465,E2 -8198.465} C_VEL
LIN {X 0,Y 453.901,Z 484.299,A -85,B 0,C 180,E1 -8199.807,E2 -8199.807} C_VEL
LIN {X 0,Y 454.235,Z 478.861,A -85,B 0,C 180,E1 -8201.152,E2 -8201.152} C_VEL
LIN {X 0,Y 454.52,Z 472.056,A -85,B 0,C 180,E1 -8202.502,E2 -8202.502} C_VEL
LIN {X 0,Y 455.115,Z 463.454,A -85,B 0,C 180,E1 -8203.849,E2 -8203.849} C_VEL
LIN {X 0,Y 455.572,Z 454.622,A -85,B 0,C 180,E1 -8204.975,E2 -8204.975} C_VEL
LIN {X 0,Y 456.054,Z 444.863,A -85,B 0,C 180,E1 -8205.99,E2 -8205.99} C_VEL
LIN {X 0,Y 456.539,Z 433.982,A -85,B 0,C 180,E1 -8206.892,E2 -8206.892} C_VEL
LIN {X 0,Y 456.755,Z 425.836,A -85,B 0,C 180,E1 -8207.448,E2 -8207.448} C_VEL
LIN {X 0,Y 453.544,Z 414.993,A -85,B 0,C 180,E1 -8208.2,E2 -8208.2} C_VEL
LIN {X 0,Y 453.485,Z 414.995,A -85,B 0,C 180,E1 -8211.585,E2 -8211.585} C_VEL
LIN {X 0,Y 453.506,Z 414.993,A -85,B 0,C 180,E1 -8214.735,E2 -8214.735} C_VEL
LIN {X 0,Y 453.537,Z 414.99,A -85,B 0,C 180,E1 -8217.96,E2 -8217.96} C_VEL
LIN {X 0,Y 453.471,Z 414.995,A -85,B 0,C 180,E1 -8221.525,E2 -8221.525} C_VEL
LIN {X 0,Y 453.494,Z 414.993,A -85,B 0,C 180,E1 -8224.778,E2 -8224.778} C_VEL
LIN {X 0,Y 453.469,Z 415,A -85,B 0,C 180,E1 -8228.312,E2 -8228.312} C_VEL
LIN {X 0,Y 453.498,Z 414.993,A -85,B 0,C 180,E1 -8230.609,E2 -8230.609} C_VEL
LIN {X 0,Y 453.46,Z 414.996,A -85,B 0,C 180,E1 -8233.244,E2 -8233.244} C_VEL
LIN {X 0,Y 453.471,Z 414.998,A -85,B 0,C 180,E1 -8235.779,E2 -8235.779} C_VEL
LIN {X 0,Y 453.484,Z 414.998,A -85,B 0,C 180,E1 -8238.209,E2 -8238.209} C_VEL
LIN {X 0,Y 453.499,Z 414.991,A -85,B 0,C 180,E1 -8240.793,E2 -8240.793} C_VEL
LIN {X 0,Y 453.459,Z 415.003,A -85,B 0,C 180,E1 -8243.917,E2 -8243.917} C_VEL
LIN {X 0,Y 453.487,Z 414.992,A -85,B 0,C 180,E1 -8247.151,E2 -8247.151} C_VEL
LIN {X 0,Y 453.479,Z 414.996,A -85,B 0,C 180,E1 -8250.268,E2 -8250.268} C_VEL
LIN {X 0,Y 453.506,Z 414.991,A -85,B 0,C 180,E1 -8253.294,E2 -8253.294} C_VEL
LIN {X 0,Y 453.502,Z 414.993,A -85,B 0,C 180,E1 -8256.238,E2 -8256.238} C_VEL
LIN {X 0,Y 453.487,Z 414.993,A -85,B 0,C 180,E1 -8259.118,E2 -8259.118} C_VEL
LIN {X 0,Y 453.509,Z 414.995,A -85,B 0,C 180,E1 -8261.944,E2 -8261.944} C_VEL
LIN {X 0,Y 453.544,Z 414.985,A -85,B 0,C 180,E1 -8264.726,E2 -8264.726} C_VEL
LIN {X 0,Y 453.564,Z 414.988,A -85,B 0,C 180,E1 -8266.274,E2 -8266.274} C_VEL
LIN {X 0,Y 456.189,Z 425.054,A -85,B 0,C 180,E1 -8266.958,E2 -8266.958} C_VEL
LIN {X 0,Y 455.695,Z 436.289,A -85,B 0,C 180,E1 -8267.757,E2 -8267.757} C_VEL
LIN {X 0,Y 455.249,Z 447.485,A -85,B 0,C 180,E1 -8268.761,E2 -8268.761} C_VEL
LIN {X 0,Y 454.949,Z 456.608,A -85,B 0,C 180,E1 -8269.767,E2 -8269.767} C_VEL
LIN {X 0,Y 454.476,Z 465.002,A -85,B 0,C 180,E1 -8270.88,E2 -8270.88} C_VEL
LIN {X 0,Y 454.066,Z 473.236,A -85,B 0,C 180,E1 -8272.227,E2 -8272.227} C_VEL
LIN {X 0,Y 453.818,Z 478.774,A -85,B 0,C 180,E1 -8273.33,E2 -8273.33} C_VEL
LIN {X 0,Y 453.484,Z 484.256,A -85,B 0,C 180,E1 -8274.664,E2 -8274.664} C_VEL
LIN {X 0,Y 453.451,Z 488.529,A -85,B 0,C 180,E1 -8276,E2 -8276} C_VEL
LIN {X 0,Y 453.147,Z 491.784,A -85,B 0,C 180,E1 -8277.333,E2 -8277.333} C_VEL
LIN {X 0,Y 453.193,Z 493.403,A -85,B 0,C 180,E1 -8278.223,E2 -8278.223} C_VEL
LIN {X 0,Y 453.111,Z 494.59,A -85,B 0,C 180,E1 -8279.111,E2 -8279.111} C_VEL
LIN {X 0,Y 453.108,Z 495.762,A -85,B 0,C 180,E1 -8280.889,E2 -8280.889} C_VEL
LIN {X 0,Y 453.184,Z 495.752,A -85,B 0,C 180,E1 -8281.777,E2 -8281.777} C_VEL
LIN {X 0,Y 453.225,Z 494.502,A -85,B 0,C 180,E1 -8283.556,E2 -8283.556} C_VEL
LIN {X 0,Y 453.312,Z 493.294,A -85,B 0,C 180,E1 -8284.446,E2 -8284.446} C_VEL
LIN {X 0,Y 453.527,Z 490.638,A -85,B 0,C 180,E1 -8285.781,E2 -8285.781} C_VEL
LIN {X 0,Y 453.778,Z 486.954,A -85,B 0,C 180,E1 -8287.117,E2 -8287.117} C_VEL
LIN {X 0,Y 454.015,Z 482.124,A -85,B 0,C 180,E1 -8288.456,E2 -8288.456} C_VEL
LIN {X 0,Y 454.437,Z 474.815,A -85,B 0,C 180,E1 -8290.019,E2 -8290.019} C_VEL
LIN {X 0,Y 454.891,Z 466.854,A -85,B 0,C 180,E1 -8291.361,E2 -8291.361} C_VEL
LIN {X 0,Y 455.266,Z 458.678,A -85,B 0,C 180,E1 -8292.481,E2 -8292.481} C_VEL
LIN {X 0,Y 455.77,Z 448.955,A -85,B 0,C 180,E1 -8293.567,E2 -8293.567} C_VEL
LIN {X 0,Y 456.323,Z 438.647,A -85,B 0,C 180,E1 -8294.494,E2 -8294.494} C_VEL
LIN {X 0,Y 456.761,Z 426.261,A -85,B 0,C 180,E1 -8295.373,E2 -8295.373} C_VEL
LIN {X 0,Y 454.15,Z 417.076,A -85,B 0,C 180,E1 -8296.018,E2 -8296.018} C_VEL
LIN {X 0,Y 453.549,Z 414.993,A -85,B 0,C 180,E1 -8296.172,E2 -8296.172} C_VEL
LIN {X 0,Y 453.522,Z 415.001,A -85,B 0,C 180,E1 -8299.04,E2 -8299.04} C_VEL
LIN {X 0,Y 453.48,Z 415.003,A -85,B 0,C 180,E1 -8301.836,E2 -8301.836} C_VEL
LIN {X 0,Y 453.504,Z 414.997,A -85,B 0,C 180,E1 -8304.735,E2 -8304.735} C_VEL
LIN {X 0,Y 453.541,Z 414.989,A -85,B 0,C 180,E1 -8307.961,E2 -8307.961} C_VEL
LIN {X 0,Y 453.469,Z 415,A -85,B 0,C 180,E1 -8311.525,E2 -8311.525} C_VEL
LIN {X 0,Y 453.491,Z 414.997,A -85,B 0,C 180,E1 -8314.777,E2 -8314.777} C_VEL
LIN {X 0,Y 453.467,Z 415.002,A -85,B 0,C 180,E1 -8318.311,E2 -8318.311} C_VEL
LIN {X 0,Y 453.497,Z 414.997,A -85,B 0,C 180,E1 -8320.609,E2 -8320.609} C_VEL
LIN {X 0,Y 453.459,Z 415.002,A -85,B 0,C 180,E1 -8323.244,E2 -8323.244} C_VEL
LIN {X 0,Y 453.469,Z 414.998,A -85,B 0,C 180,E1 -8325.779,E2 -8325.779} C_VEL
LIN {X 0,Y 453.51,Z 415.03,A -85,B 0,C 180,E1 -8328.887,E2 -8328.887} C_VEL
LIN {X 0,Y 455.497,Z 424.946,A -85,B 0,C 180,E1 -8331.896,E2 -8331.896} C_VEL
LIN {X 0,Y 456.308,Z 429.52,A -85,B 0,C 180,E1 -8333.216,E2 -8333.216} C_VEL
LIN {X 0,Y 456.035,Z 435.268,A -85,B 0,C 180,E1 -8334.765,E2 -8334.765} C_VEL
LIN {X 0,Y 455.338,Z 448.119,A -85,B 0,C 180,E1 -8338.093,E2 -8338.093} C_VEL
LIN {X 0,Y 454.746,Z 461.265,A -85,B 0,C 180,E1 -8341.373,E2 -8341.373} C_VEL
LIN {X 0,Y 454.239,Z 474.437,A -85,B 0,C 180,E1 -8344.573,E2 -8344.573} C_VEL
LIN {X 0,Y 453.799,Z 488.537,A -85,B 0,C 180,E1 -8347.941,E2 -8347.941} C_VEL
LIN {X 0,Y 453.384,Z 503.474,A -85,B 0,C 180,E1 -8351.471,E2 -8351.471} C_VEL
LIN {X 0,Y 453.16,Z 514.267,A -85,B 0,C 180,E1 -8354.023,E2 -8354.023} C_VEL
LIN {X 0,Y 454.599,Z 528.372,A -85,B 0,C 180,E1 -8354.422,E2 -8354.422} C_VEL
LIN {X 0,Y 455.532,Z 540.273,A -85,B 0,C 180,E1 -8354.909,E2 -8354.909} C_VEL
LIN {X 0,Y 455.716,Z 545.031,A -85,B 0,C 180,E1 -8355.144,E2 -8355.144} C_VEL
LIN {X 0,Y 455.154,Z 556.716,A -85,B 0,C 180,E1 -8355.811,E2 -8355.811} C_VEL
LIN {X 0,Y 454.542,Z 568.62,A -85,B 0,C 180,E1 -8356.693,E2 -8356.693} C_VEL
LIN {X 0,Y 454.087,Z 579.514,A -85,B 0,C 180,E1 -8357.713,E2 -8357.713} C_VEL
LIN {X 0,Y 453.564,Z 589.249,A -85,B 0,C 180,E1 -8358.832,E2 -8358.832} C_VEL
LIN {X 0,Y 453.159,Z 598.67,A -85,B 0,C 180,E1 -8360.177,E2 -8360.177} C_VEL
LIN {X 0,Y 452.957,Z 606.279,A -85,B 0,C 180,E1 -8361.523,E2 -8361.523} C_VEL
LIN {X 0,Y 452.863,Z 612.414,A -85,B 0,C 180,E1 -8362.868,E2 -8362.868} C_VEL
LIN {X 0,Y 452.854,Z 617.28,A -85,B 0,C 180,E1 -8364.21,E2 -8364.21} C_VEL
LIN {X 0,Y 452.871,Z 621.006,A -85,B 0,C 180,E1 -8365.55,E2 -8365.55} C_VEL
LIN {X 0,Y 452.881,Z 622.931,A -85,B 0,C 180,E1 -8366.441,E2 -8366.441} C_VEL
LIN {X 0,Y 452.874,Z 624.374,A -85,B 0,C 180,E1 -8367.331,E2 -8367.331} C_VEL
LIN {X 0,Y 453.004,Z 626.056,A -85,B 0,C 180,E1 -8369.111,E2 -8369.111} C_VEL
LIN {X 0,Y 452.993,Z 626.279,A -85,B 0,C 180,E1 -8370,E2 -8370} C_VEL
LIN {X 0,Y 453.004,Z 626.059,A -85,B 0,C 180,E1 -8370.889,E2 -8370.889} C_VEL
LIN {X 0,Y 452.873,Z 624.389,A -85,B 0,C 180,E1 -8372.668,E2 -8372.668} C_VEL
LIN {X 0,Y 452.877,Z 622.945,A -85,B 0,C 180,E1 -8373.559,E2 -8373.559} C_VEL
LIN {X 0,Y 452.864,Z 619.911,A -85,B 0,C 180,E1 -8374.896,E2 -8374.896} C_VEL
LIN {X 0,Y 452.847,Z 615.801,A -85,B 0,C 180,E1 -8376.237,E2 -8376.237} C_VEL
LIN {X 0,Y 452.904,Z 609.488,A -85,B 0,C 180,E1 -8377.804,E2 -8377.804} C_VEL
LIN {X 0,Y 453.065,Z 602.616,A -85,B 0,C 180,E1 -8379.149,E2 -8379.149} C_VEL
LIN {X 0,Y 453.331,Z 594.108,A -85,B 0,C 180,E1 -8380.495,E2 -8380.495} C_VEL
LIN {X 0,Y 453.712,Z 585.397,A -85,B 0,C 180,E1 -8381.617,E2 -8381.617} C_VEL
LIN {X 0,Y 454.193,Z 575.874,A -85,B 0,C 180,E1 -8382.624,E2 -8382.624} C_VEL
LIN {X 0,Y 454.781,Z 564.084,A -85,B 0,C 180,E1 -8383.631,E2 -8383.631} C_VEL
LIN {X 0,Y 455.306,Z 552.464,A -85,B 0,C 180,E1 -8384.412,E2 -8384.412} C_VEL
LIN {X 0,Y 455.687,Z 541.751,A -85,B 0,C 180,E1 -8384.971,E2 -8384.971} C_VEL
LIN {X 0,Y 454.648,Z 530.535,A -85,B 0,C 180,E1 -8385.448,E2 -8385.448} C_VEL
LIN {X 0,Y 453.413,Z 517.338,A -85,B 0,C 180,E1 -8385.837,E2 -8385.837} C_VEL
LIN {X 0,Y 453.138,Z 514.444,A -85,B 0,C 180,E1 -8385.908,E2 -8385.908} C_VEL
LIN {X 0,Y 453.428,Z 501.224,A -85,B 0,C 180,E1 -8389.006,E2 -8389.006} C_VEL
LIN {X 0,Y 453.787,Z 487.186,A -85,B 0,C 180,E1 -8392.299,E2 -8392.299} C_VEL
LIN {X 0,Y 454.242,Z 472.904,A -85,B 0,C 180,E1 -8395.672,E2 -8395.672} C_VEL
LIN {X 0,Y 454.773,Z 458.504,A -85,B 0,C 180,E1 -8399.13,E2 -8399.13} C_VEL
LIN {X 0,Y 455.282,Z 445.881,A -85,B 0,C 180,E1 -8402.24,E2 -8402.24} C_VEL
LIN {X 0,Y 456.023,Z 431.713,A -85,B 0,C 180,E1 -8405.848,E2 -8405.848} C_VEL
LIN {X 0,Y 455.916,Z 427.586,A -85,B 0,C 180,E1 -8406.955,E2 -8406.955} C_VEL
LIN {X 0,Y 453.979,Z 417.123,A -85,B 0,C 180,E1 -8409.973,E2 -8409.973} C_VEL
LIN {X 0,Y 453.543,Z 414.993,A -85,B 0,C 180,E1 -8410.677,E2 -8410.677} C_VEL
LIN {X 0,Y 453.467,Z 415.004,A -85,B 0,C 180,E1 -8414.221,E2 -8414.221} C_VEL
LIN {X 0,Y 453.47,Z 415.004,A -85,B 0,C 180,E1 -8417.006,E2 -8417.006} C_VEL
LIN {X 0,Y 453.518,Z 414.995,A -85,B 0,C 180,E1 -8420.553,E2 -8420.553} C_VEL
LIN {X 0,Y 453.457,Z 415.002,A -85,B 0,C 180,E1 -8423.917,E2 -8423.917} C_VEL
LIN {X 0,Y 453.484,Z 414.996,A -85,B 0,C 180,E1 -8427.151,E2 -8427.151} C_VEL
LIN {X 0,Y 453.476,Z 415,A -85,B 0,C 180,E1 -8430.268,E2 -8430.268} C_VEL
LIN {X 0,Y 453.515,Z 414.993,A -85,B 0,C 180,E1 -8433.294,E2 -8433.294} C_VEL
LIN {X 0,Y 453.505,Z 414.998,A -85,B 0,C 180,E1 -8436.239,E2 -8436.239} C_VEL
LIN {X 0,Y 453.484,Z 414.996,A -85,B 0,C 180,E1 -8439.118,E2 -8439.118} C_VEL
LIN {X 0,Y 453.514,Z 414.997,A -85,B 0,C 180,E1 -8441.945,E2 -8441.945} C_VEL
LIN {X 0,Y 453.541,Z 414.991,A -85,B 0,C 180,E1 -8444.726,E2 -8444.726} C_VEL
LIN {X 0,Y 453.603,Z 414.983,A -85,B 0,C 180,E1 -8447.472,E2 -8447.472} C_VEL
LIN {X 0,Y 453.588,Z 414.983,A -85,B 0,C 180,E1 -8451.087,E2 -8451.087} C_VEL
LIN {X 0,Y 453.675,Z 414.975,A -85,B 0,C 180,E1 -8453.775,E2 -8453.775} C_VEL
LIN {X 0,Y 453.769,Z 414.962,A -85,B 0,C 180,E1 -8457.337,E2 -8457.337} C_VEL
LIN {X 0,Y 453.826,Z 414.957,A -85,B 0,C 180,E1 -8460,E2 -8460} C_VEL
LIN {X 0,Y 453.746,Z 414.964,A -85,B 0,C 180,E1 -8462.663,E2 -8462.663} C_VEL
LIN {X 0,Y 453.679,Z 414.975,A -85,B 0,C 180,E1 -8466.225,E2 -8466.225} C_VEL
LIN {X 0,Y 453.595,Z 414.983,A -85,B 0,C 180,E1 -8468.914,E2 -8468.914} C_VEL
LIN {X 0,Y 453.565,Z 414.988,A -85,B 0,C 180,E1 -8472.529,E2 -8472.529} C_VEL
LIN {X 0,Y 453.546,Z 414.992,A -85,B 0,C 180,E1 -8476.196,E2 -8476.196} C_VEL
LIN {X 0,Y 453.523,Z 414.992,A -85,B 0,C 180,E1 -8479.041,E2 -8479.041} C_VEL
LIN {X 0,Y 453.479,Z 415.001,A -85,B 0,C 180,E1 -8481.836,E2 -8481.836} C_VEL
LIN {X 0,Y 453.516,Z 414.993,A -85,B 0,C 180,E1 -8484.735,E2 -8484.735} C_VEL
LIN {X 0,Y 453.539,Z 414.993,A -85,B 0,C 180,E1 -8487.961,E2 -8487.961} C_VEL
LIN {X 0,Y 453.468,Z 415.001,A -85,B 0,C 180,E1 -8491.525,E2 -8491.525} C_VEL
LIN {X 0,Y 453.491,Z 414.996,A -85,B 0,C 180,E1 -8494.778,E2 -8494.778} C_VEL
LIN {X 0,Y 453.475,Z 414.999,A -85,B 0,C 180,E1 -8498.311,E2 -8498.311} C_VEL
LIN {X 0,Y 453.496,Z 414.994,A -85,B 0,C 180,E1 -8500.609,E2 -8500.609} C_VEL
LIN {X 0,Y 453.466,Z 415,A -85,B 0,C 180,E1 -8503.246,E2 -8503.246} C_VEL
LIN {X 0,Y 453.476,Z 415.002,A -85,B 0,C 180,E1 -8505.78,E2 -8505.78} C_VEL
LIN {X 0,Y 453.484,Z 414.998,A -85,B 0,C 180,E1 -8508.21,E2 -8508.21} C_VEL
LIN {X 0,Y 453.513,Z 414.993,A -85,B 0,C 180,E1 -8510.791,E2 -8510.791} C_VEL
LIN {X 0,Y 453.46,Z 415.003,A -85,B 0,C 180,E1 -8513.918,E2 -8513.918} C_VEL
LIN {X 0,Y 453.487,Z 414.997,A -85,B 0,C 180,E1 -8517.152,E2 -8517.152} C_VEL
LIN {X 0,Y 453.518,Z 414.994,A -85,B 0,C 180,E1 -8520.271,E2 -8520.271} C_VEL
LIN {X 0,Y 453.513,Z 414.995,A -85,B 0,C 180,E1 -8523.294,E2 -8523.294} C_VEL
LIN {X 0,Y 453.507,Z 414.995,A -85,B 0,C 180,E1 -8526.239,E2 -8526.239} C_VEL
LIN {X 0,Y 453.487,Z 414.997,A -85,B 0,C 180,E1 -8529.118,E2 -8529.118} C_VEL
LIN {X 0,Y 453.516,Z 414.995,A -85,B 0,C 180,E1 -8531.945,E2 -8531.945} C_VEL
LIN {X 0,Y 453.544,Z 414.992,A -85,B 0,C 180,E1 -8534.727,E2 -8534.727} C_VEL
LIN {X 0,Y 453.611,Z 414.981,A -85,B 0,C 180,E1 -8538.01,E2 -8538.01} C_VEL
LIN {X 0,Y 456.642,Z 426.637,A -85,B 0,C 180,E1 -8538.796,E2 -8538.796} C_VEL
LIN {X 0,Y 456.207,Z 438.956,A -85,B 0,C 180,E1 -8539.684,E2 -8539.684} C_VEL
LIN {X 0,Y 456.063,Z 441.369,A -85,B 0,C 180,E1 -8539.887,E2 -8539.887} C_VEL
LIN {X 0,Y 455.154,Z 446.267,A -85,B 0,C 180,E1 -8540.303,E2 -8540.303} C_VEL
LIN {X 0,Y 451.909,Z 453.985,A -85,B 0,C 180,E1 -8540.986,E2 -8540.986} C_VEL
LIN {X 0,Y 448.756,Z 461.169,A -85,B 0,C 180,E1 -8541.748,E2 -8541.748} C_VEL
LIN {X 0,Y 447.985,Z 465.179,A -85,B 0,C 180,E1 -8542.281,E2 -8542.281} C_VEL
LIN {X 0,Y 447.589,Z 472.561,A -85,B 0,C 180,E1 -8543.464,E2 -8543.464} C_VEL
LIN {X 0,Y 447.088,Z 479.45,A -85,B 0,C 180,E1 -8544.814,E2 -8544.814} C_VEL
LIN {X 0,Y 446.736,Z 485.708,A -85,B 0,C 180,E1 -8546.392,E2 -8546.392} C_VEL
LIN {X 0,Y 446.574,Z 489.831,A -85,B 0,C 180,E1 -8547.745,E2 -8547.745} C_VEL
LIN {X 0,Y 446.313,Z 492.951,A -85,B 0,C 180,E1 -8549.098,E2 -8549.098} C_VEL
LIN {X 0,Y 446.245,Z 494.496,A -85,B 0,C 180,E1 -8550,E2 -8550} C_VEL
LIN {X 0,Y 446.092,Z 495.665,A -85,B 0,C 180,E1 -8550.903,E2 -8550.903} C_VEL
LIN {X 0,Y 446.16,Z 496.378,A -85,B 0,C 180,E1 -8551.806,E2 -8551.806} C_VEL
LIN {X 0,Y 446.107,Z 496.717,A -85,B 0,C 180,E1 -8553.613,E2 -8553.613} C_VEL
LIN {X 0,Y 446.168,Z 496.321,A -85,B 0,C 180,E1 -8554.517,E2 -8554.517} C_VEL
LIN {X 0,Y 446.304,Z 495.495,A -85,B 0,C 180,E1 -8555.422,E2 -8555.422} C_VEL
LIN {X 0,Y 446.451,Z 492.697,A -85,B 0,C 180,E1 -8557.235,E2 -8557.235} C_VEL
LIN {X 0,Y 446.618,Z 489.48,A -85,B 0,C 180,E1 -8558.598,E2 -8558.598} C_VEL
LIN {X 0,Y 446.961,Z 485.191,A -85,B 0,C 180,E1 -8559.96,E2 -8559.96} C_VEL
LIN {X 0,Y 447.314,Z 479.725,A -85,B 0,C 180,E1 -8561.326,E2 -8561.326} C_VEL
LIN {X 0,Y 447.629,Z 472.872,A -85,B 0,C 180,E1 -8562.698,E2 -8562.698} C_VEL
LIN {X 0,Y 448.265,Z 464.226,A -85,B 0,C 180,E1 -8564.065,E2 -8564.065} C_VEL
LIN {X 0,Y 448.788,Z 454.379,A -85,B 0,C 180,E1 -8565.323,E2 -8565.323} C_VEL
LIN {X 0,Y 449.349,Z 444.244,A -85,B 0,C 180,E1 -8566.352,E2 -8566.352} C_VEL
LIN {X 0,Y 449.816,Z 432.959,A -85,B 0,C 180,E1 -8567.269,E2 -8567.269} C_VEL
LIN {X 0,Y 449.905,Z 427.317,A -85,B 0,C 180,E1 -8567.657,E2 -8567.657} C_VEL
LIN {X 0,Y 446.516,Z 415.869,A -85,B 0,C 180,E1 -8568.459,E2 -8568.459} C_VEL
LIN {X 0,Y 446.453,Z 415.872,A -85,B 0,C 180,E1 -8571.755,E2 -8571.755} C_VEL
LIN {X 0,Y 446.449,Z 415.869,A -85,B 0,C 180,E1 -8575.153,E2 -8575.153} C_VEL
LIN {X 0,Y 446.489,Z 415.87,A -85,B 0,C 180,E1 -8578.179,E2 -8578.179} C_VEL
LIN {X 0,Y 446.424,Z 415.874,A -85,B 0,C 180,E1 -8581.775,E2 -8581.775} C_VEL
LIN {X 0,Y 446.436,Z 415.874,A -85,B 0,C 180,E1 -8584.523,E2 -8584.523} C_VEL
LIN {X 0,Y 446.421,Z 415.879,A -85,B 0,C 180,E1 -8588.079,E2 -8588.079} C_VEL
LIN {X 0,Y 446.431,Z 415.871,A -85,B 0,C 180,E1 -8590.918,E2 -8590.918} C_VEL
LIN {X 0,Y 446.406,Z 415.879,A -85,B 0,C 180,E1 -8593.846,E2 -8593.846} C_VEL
LIN {X 0,Y 446.404,Z 415.878,A -85,B 0,C 180,E1 -8596.403,E2 -8596.403} C_VEL
LIN {X 0,Y 446.431,Z 415.871,A -85,B 0,C 180,E1 -8599.082,E2 -8599.082} C_VEL
LIN {X 0,Y 446.414,Z 415.879,A -85,B 0,C 180,E1 -8602.121,E2 -8602.121} C_VEL
LIN {X 0,Y 446.433,Z 415.873,A -85,B 0,C 180,E1 -8605.477,E2 -8605.477} C_VEL
LIN {X 0,Y 446.42,Z 415.873,A -85,B 0,C 180,E1 -8608.7,E2 -8608.7} C_VEL
LIN {X 0,Y 446.489,Z 415.871,A -85,B 0,C 180,E1 -8611.821,E2 -8611.821} C_VEL
LIN {X 0,Y 446.449,Z 415.869,A -85,B 0,C 180,E1 -8614.847,E2 -8614.847} C_VEL
LIN {X 0,Y 446.453,Z 415.871,A -85,B 0,C 180,E1 -8618.245,E2 -8618.245} C_VEL
LIN {X 0,Y 446.457,Z 415.875,A -85,B 0,C 180,E1 -8621.649,E2 -8621.649} C_VEL
LIN {X 0,Y 446.512,Z 415.861,A -85,B 0,C 180,E1 -8624.48,E2 -8624.48} C_VEL
LIN {X 0,Y 446.549,Z 415.99,A -85,B 0,C 180,E1 -8626.098,E2 -8626.098} C_VEL
LIN {X 0,Y 449.201,Z 425.959,A -85,B 0,C 180,E1 -8626.776,E2 -8626.776} C_VEL
LIN {X 0,Y 448.804,Z 436.903,A -85,B 0,C 180,E1 -8627.566,E2 -8627.566} C_VEL
LIN {X 0,Y 448.318,Z 448.154,A -85,B 0,C 180,E1 -8628.585,E2 -8628.585} C_VEL
LIN {X 0,Y 448.012,Z 457.326,A -85,B 0,C 180,E1 -8629.607,E2 -8629.607} C_VEL
LIN {X 0,Y 447.519,Z 465.779,A -85,B 0,C 180,E1 -8630.737,E2 -8630.737} C_VEL
LIN {X 0,Y 447.075,Z 474.199,A -85,B 0,C 180,E1 -8632.131,E2 -8632.131} C_VEL
LIN {X 0,Y 446.774,Z 480.647,A -85,B 0,C 180,E1 -8633.451,E2 -8633.451} C_VEL
LIN {X 0,Y 446.501,Z 486.725,A -85,B 0,C 180,E1 -8635.033,E2 -8635.033} C_VEL
LIN {X 0,Y 446.249,Z 490.692,A -85,B 0,C 180,E1 -8636.388,E2 -8636.388} C_VEL
LIN {X 0,Y 446.122,Z 492.751,A -85,B 0,C 180,E1 -8637.291,E2 -8637.291} C_VEL
LIN {X 0,Y 446.175,Z 494.387,A -85,B 0,C 180,E1 -8638.195,E2 -8638.195} C_VEL
LIN {X 0,Y 446.091,Z 495.592,A -85,B 0,C 180,E1 -8639.097,E2 -8639.097} C_VEL
LIN {X 0,Y 446.088,Z 496.794,A -85,B 0,C 180,E1 -8640.903,E2 -8640.903} C_VEL
LIN {X 0,Y 446.167,Z 496.796,A -85,B 0,C 180,E1 -8641.805,E2 -8641.805} C_VEL
LIN {X 0,Y 446.216,Z 495.566,A -85,B 0,C 180,E1 -8643.612,E2 -8643.612} C_VEL
LIN {X 0,Y 446.312,Z 494.363,A -85,B 0,C 180,E1 -8644.516,E2 -8644.516} C_VEL
LIN {X 0,Y 446.545,Z 491.713,A -85,B 0,C 180,E1 -8645.872,E2 -8645.872} C_VEL
LIN {X 0,Y 446.824,Z 488.044,A -85,B 0,C 180,E1 -8647.229,E2 -8647.229} C_VEL
LIN {X 0,Y 447.08,Z 483.243,A -85,B 0,C 180,E1 -8648.588,E2 -8648.588} C_VEL
LIN {X 0,Y 447.537,Z 475.98,A -85,B 0,C 180,E1 -8650.176,E2 -8650.176} C_VEL
LIN {X 0,Y 448.031,Z 468.043,A -85,B 0,C 180,E1 -8651.537,E2 -8651.537} C_VEL
LIN {X 0,Y 448.437,Z 459.876,A -85,B 0,C 180,E1 -8652.674,E2 -8652.674} C_VEL
LIN {X 0,Y 448.937,Z 450.851,A -85,B 0,C 180,E1 -8653.705,E2 -8653.705} C_VEL
LIN {X 0,Y 449.565,Z 439.877,A -85,B 0,C 180,E1 -8654.716,E2 -8654.716} C_VEL
LIN {X 0,Y 450.02,Z 428.098,A -85,B 0,C 180,E1 -8655.574,E2 -8655.574} C_VEL
LIN {X 0,Y 447.953,Z 420.437,A -85,B 0,C 180,E1 -8656.144,E2 -8656.144} C_VEL
LIN {X 0,Y 446.493,Z 415.87,A -85,B 0,C 180,E1 -8656.459,E2 -8656.459} C_VEL
LIN {X 0,Y 446.473,Z 415.878,A -85,B 0,C 180,E1 -8659.303,E2 -8659.303} C_VEL
LIN {X 0,Y 446.421,Z 415.881,A -85,B 0,C 180,E1 -8662.199,E2 -8662.199} C_VEL
LIN {X 0,Y 446.448,Z 415.875,A -85,B 0,C 180,E1 -8665.153,E2 -8665.153} C_VEL
LIN {X 0,Y 446.488,Z 415.868,A -85,B 0,C 180,E1 -8668.178,E2 -8668.178} C_VEL
LIN {X 0,Y 446.423,Z 415.877,A -85,B 0,C 180,E1 -8671.775,E2 -8671.775} C_VEL
LIN {X 0,Y 446.432,Z 415.877,A -85,B 0,C 180,E1 -8674.523,E2 -8674.523} C_VEL
LIN {X 0,Y 446.419,Z 415.878,A -85,B 0,C 180,E1 -8678.079,E2 -8678.079} C_VEL
LIN {X 0,Y 446.431,Z 415.877,A -85,B 0,C 180,E1 -8680.918,E2 -8680.918} C_VEL
LIN {X 0,Y 446.405,Z 415.878,A -85,B 0,C 180,E1 -8683.846,E2 -8683.846} C_VEL
LIN {X 0,Y 446.403,Z 415.879,A -85,B 0,C 180,E1 -8686.403,E2 -8686.403} C_VEL
LIN {X 0,Y 446.477,Z 416.059,A -85,B 0,C 180,E1 -8688.614,E2 -8688.614} C_VEL
LIN {X 0,Y 448.423,Z 425.674,A -85,B 0,C 180,E1 -8691.595,E2 -8691.595} C_VEL
LIN {X 0,Y 449.401,Z 431.233,A -85,B 0,C 180,E1 -8693.236,E2 -8693.236} C_VEL
LIN {X 0,Y 448.954,Z 438.308,A -85,B 0,C 180,E1 -8695.153,E2 -8695.153} C_VEL
LIN {X 0,Y 448.281,Z 450.435,A -85,B 0,C 180,E1 -8698.33,E2 -8698.33} C_VEL
LIN {X 0,Y 447.677,Z 463.082,A -85,B 0,C 180,E1 -8701.538,E2 -8701.538} C_VEL
LIN {X 0,Y 447.169,Z 475.628,A -85,B 0,C 180,E1 -8704.641,E2 -8704.641} C_VEL
LIN {X 0,Y 446.746,Z 488.669,A -85,B 0,C 180,E1 -8707.817,E2 -8707.817} C_VEL
LIN {X 0,Y 446.298,Z 504.508,A -85,B 0,C 180,E1 -8711.642,E2 -8711.642} C_VEL
LIN {X 0,Y 446.078,Z 513.219,A -85,B 0,C 180,E1 -8713.741,E2 -8713.741} C_VEL
LIN {X 0,Y 447.603,Z 527.863,A -85,B 0,C 180,E1 -8714.175,E2 -8714.175} C_VEL
LIN {X 0,Y 448.451,Z 539.527,A -85,B 0,C 180,E1 -8714.665,E2 -8714.665} C_VEL
LIN {X 0,Y 448.832,Z 544.261,A -85,B 0,C 180,E1 -8714.911,E2 -8714.911} C_VEL
LIN {X 0,Y 448.234,Z 555.882,A -85,B 0,C 180,E1 -8715.587,E2 -8715.587} C_VEL
LIN {X 0,Y 447.584,Z 567.686,A -85,B 0,C 180,E1 -8716.479,E2 -8716.479} C_VEL
LIN {X 0,Y 447.068,Z 578.591,A -85,B 0,C 180,E1 -8717.517,E2 -8717.517} C_VEL
LIN {X 0,Y 446.541,Z 588.306,A -85,B 0,C 180,E1 -8718.654,E2 -8718.654} C_VEL
LIN {X 0,Y 446.094,Z 597.701,A -85,B 0,C 180,E1 -8720.02,E2 -8720.02} C_VEL
LIN {X 0,Y 445.877,Z 605.298,A -85,B 0,C 180,E1 -8721.388,E2 -8721.388} C_VEL
LIN {X 0,Y 445.779,Z 611.424,A -85,B 0,C 180,E1 -8722.754,E2 -8722.754} C_VEL
LIN {X 0,Y 445.795,Z 616.286,A -85,B 0,C 180,E1 -8724.118,E2 -8724.118} C_VEL
LIN {X 0,Y 445.823,Z 620.009,A -85,B 0,C 180,E1 -8725.479,E2 -8725.479} C_VEL
LIN {X 0,Y 445.838,Z 621.929,A -85,B 0,C 180,E1 -8726.385,E2 -8726.385} C_VEL
LIN {X 0,Y 445.831,Z 623.368,A -85,B 0,C 180,E1 -8727.289,E2 -8727.289} C_VEL
LIN {X 0,Y 445.986,Z 625.049,A -85,B 0,C 180,E1 -8729.097,E2 -8729.097} C_VEL
LIN {X 0,Y 445.976,Z 625.268,A -85,B 0,C 180,E1 -8730,E2 -8730} C_VEL
LIN {X 0,Y 445.985,Z 625.044,A -85,B 0,C 180,E1 -8730.903,E2 -8730.903} C_VEL
LIN {X 0,Y 445.832,Z 623.364,A -85,B 0,C 180,E1 -8732.71,E2 -8732.71} C_VEL
LIN {X 0,Y 445.835,Z 621.914,A -85,B 0,C 180,E1 -8733.615,E2 -8733.615} C_VEL
LIN {X 0,Y 445.816,Z 618.871,A -85,B 0,C 180,E1 -8734.974,E2 -8734.974} C_VEL
LIN {X 0,Y 445.758,Z 613.634,A -85,B 0,C 180,E1 -8736.643,E2 -8736.643} C_VEL
LIN {X 0,Y 445.861,Z 607.378,A -85,B 0,C 180,E1 -8738.156,E2 -8738.156} C_VEL
LIN {X 0,Y 446.035,Z 600.257,A -85,B 0,C 180,E1 -8739.523,E2 -8739.523} C_VEL
LIN {X 0,Y 446.368,Z 591.36,A -85,B 0,C 180,E1 -8740.891,E2 -8740.891} C_VEL
LIN {X 0,Y 446.823,Z 582.28,A -85,B 0,C 180,E1 -8742.029,E2 -8742.029} C_VEL
LIN {X 0,Y 447.31,Z 571.735,A -85,B 0,C 180,E1 -8743.109,E2 -8743.109} C_VEL
LIN {X 0,Y 447.947,Z 559.823,A -85,B 0,C 180,E1 -8744.074,E2 -8744.074} C_VEL
LIN {X 0,Y 448.623,Z 547.22,A -85,B 0,C 180,E1 -8744.864,E2 -8744.864} C_VEL
LIN {X 0,Y 448.588,Z 541.604,A -85,B 0,C 180,E1 -8745.156,E2 -8745.156} C_VEL
LIN {X 0,Y 447.609,Z 530.023,A -85,B 0,C 180,E1 -8745.664,E2 -8745.664} C_VEL
LIN {X 0,Y 446.387,Z 516.862,A -85,B 0,C 180,E1 -8746.067,E2 -8746.067} C_VEL
LIN {X 0,Y 446.092,Z 513.368,A -85,B 0,C 180,E1 -8746.168,E2 -8746.168} C_VEL
LIN {X 0,Y 446.422,Z 499.238,A -85,B 0,C 180,E1 -8749.544,E2 -8749.544} C_VEL
LIN {X 0,Y 446.798,Z 485.189,A -85,B 0,C 180,E1 -8752.911,E2 -8752.911} C_VEL
LIN {X 0,Y 447.255,Z 471.954,A -85,B 0,C 180,E1 -8756.103,E2 -8756.103} C_VEL
LIN {X 0,Y 447.799,Z 457.584,A -85,B 0,C 180,E1 -8759.629,E2 -8759.629} C_VEL
LIN {X 0,Y 448.345,Z 445.236,A -85,B 0,C 180,E1 -8762.738,E2 -8762.738} C_VEL
LIN {X 0,Y 449.13,Z 431.893,A -85,B 0,C 180,E1 -8766.21,E2 -8766.21} C_VEL
LIN {X 0,Y 448.578,Z 426.696,A -85,B 0,C 180,E1 -8767.664,E2 -8767.664} C_VEL
LIN {X 0,Y 446.729,Z 417.04,A -85,B 0,C 180,E1 -8770.534,E2 -8770.534} C_VEL
LIN {X 0,Y 446.477,Z 415.873,A -85,B 0,C 180,E1 -8770.925,E2 -8770.925} C_VEL
LIN {X 0,Y 446.403,Z 415.882,A -85,B 0,C 180,E1 -8773.846,E2 -8773.846} C_VEL
LIN {X 0,Y 446.422,Z 415.879,A -85,B 0,C 180,E1 -8776.4,E2 -8776.4} C_VEL
LIN {X 0,Y 446.452,Z 415.874,A -85,B 0,C 180,E1 -8779.803,E2 -8779.803} C_VEL
LIN {X 0,Y 446.429,Z 415.878,A -85,B 0,C 180,E1 -8782.123,E2 -8782.123} C_VEL
LIN {X 0,Y 446.431,Z 415.875,A -85,B 0,C 180,E1 -8785.477,E2 -8785.477} C_VEL
LIN {X 0,Y 446.417,Z 415.878,A -85,B 0,C 180,E1 -8788.7,E2 -8788.7} C_VEL
LIN {X 0,Y 446.485,Z 415.87,A -85,B 0,C 180,E1 -8791.821,E2 -8791.821} C_VEL
LIN {X 0,Y 446.46,Z 415.872,A -85,B 0,C 180,E1 -8794.848,E2 -8794.848} C_VEL
LIN {X 0,Y 446.449,Z 415.876,A -85,B 0,C 180,E1 -8798.245,E2 -8798.245} C_VEL
LIN {X 0,Y 446.459,Z 415.873,A -85,B 0,C 180,E1 -8801.649,E2 -8801.649} C_VEL
LIN {X 0,Y 446.509,Z 415.868,A -85,B 0,C 180,E1 -8804.48,E2 -8804.48} C_VEL
LIN {X 0,Y 446.541,Z 415.866,A -85,B 0,C 180,E1 -8808.194,E2 -8808.194} C_VEL
LIN {X 0,Y 446.535,Z 415.861,A -85,B 0,C 180,E1 -8810.945,E2 -8810.945} C_VEL
LIN {X 0,Y 446.643,Z 415.85,A -85,B 0,C 180,E1 -8813.676,E2 -8813.676} C_VEL
LIN {X 0,Y 446.713,Z 415.84,A -85,B 0,C 180,E1 -8817.295,E2 -8817.295} C_VEL
LIN {X 0,Y 446.796,Z 415.833,A -85,B 0,C 180,E1 -8820,E2 -8820} C_VEL
LIN {X 0,Y 446.693,Z 415.843,A -85,B 0,C 180,E1 -8822.706,E2 -8822.706} C_VEL
LIN {X 0,Y 446.648,Z 415.851,A -85,B 0,C 180,E1 -8826.324,E2 -8826.324} C_VEL
LIN {X 0,Y 446.54,Z 415.861,A -85,B 0,C 180,E1 -8829.055,E2 -8829.055} C_VEL
LIN {X 0,Y 446.523,Z 415.864,A -85,B 0,C 180,E1 -8832.73,E2 -8832.73} C_VEL
LIN {X 0,Y 446.498,Z 415.87,A -85,B 0,C 180,E1 -8836.228,E2 -8836.228} C_VEL
LIN {X 0,Y 446.472,Z 415.871,A -85,B 0,C 180,E1 -8839.303,E2 -8839.303} C_VEL
LIN {X 0,Y 446.421,Z 415.879,A -85,B 0,C 180,E1 -8842.2,E2 -8842.2} C_VEL
LIN {X 0,Y 446.46,Z 415.872,A -85,B 0,C 180,E1 -8845.152,E2 -8845.152} C_VEL
LIN {X 0,Y 446.486,Z 415.871,A -85,B 0,C 180,E1 -8848.179,E2 -8848.179} C_VEL
LIN {X 0,Y 446.421,Z 415.88,A -85,B 0,C 180,E1 -8851.775,E2 -8851.775} C_VEL
LIN {X 0,Y 446.433,Z 415.876,A -85,B 0,C 180,E1 -8854.523,E2 -8854.523} C_VEL
LIN {X 0,Y 446.433,Z 415.878,A -85,B 0,C 180,E1 -8858.082,E2 -8858.082} C_VEL
LIN {X 0,Y 446.43,Z 415.874,A -85,B 0,C 180,E1 -8860.918,E2 -8860.918} C_VEL
LIN {X 0,Y 446.425,Z 415.879,A -85,B 0,C 180,E1 -8863.843,E2 -8863.843} C_VEL
LIN {X 0,Y 446.423,Z 415.877,A -85,B 0,C 180,E1 -8866.401,E2 -8866.401} C_VEL
LIN {X 0,Y 446.451,Z 415.876,A -85,B 0,C 180,E1 -8869.803,E2 -8869.803} C_VEL
LIN {X 0,Y 446.431,Z 415.877,A -85,B 0,C 180,E1 -8872.123,E2 -8872.123} C_VEL
LIN {X 0,Y 446.434,Z 415.877,A -85,B 0,C 180,E1 -8875.478,E2 -8875.478} C_VEL
LIN {X 0,Y 446.424,Z 415.876,A -85,B 0,C 180,E1 -8878.7,E2 -8878.7} C_VEL
LIN {X 0,Y 446.488,Z 415.872,A -85,B 0,C 180,E1 -8881.822,E2 -8881.822} C_VEL
LIN {X 0,Y 446.461,Z 415.87,A -85,B 0,C 180,E1 -8884.848,E2 -8884.848} C_VEL
LIN {X 0,Y 446.452,Z 415.874,A -85,B 0,C 180,E1 -8888.245,E2 -8888.245} C_VEL
LIN {X 0,Y 446.462,Z 415.875,A -85,B 0,C 180,E1 -8891.65,E2 -8891.65} C_VEL
LIN {X 0,Y 446.512,Z 415.866,A -85,B 0,C 180,E1 -8894.48,E2 -8894.48} C_VEL
LIN {X 0,Y 446.559,Z 415.86,A -85,B 0,C 180,E1 -8897.785,E2 -8897.785} C_VEL
LIN {X 0,Y 449.515,Z 426.507,A -85,B 0,C 180,E1 -8898.502,E2 -8898.502} C_VEL
LIN {X 0,Y 449.74,Z 429.898,A -85,B 0,C 180,E1 -8898.736,E2 -8898.736} C_VEL
LIN {X 0,Y 449.32,Z 440.387,A -85,B 0,C 180,E1 -8899.524,E2 -8899.524} C_VEL
LIN {X 0,Y 448.827,Z 450.472,A -85,B 0,C 180,E1 -8900.47,E2 -8900.47} C_VEL
LIN {X 0,Y 448.287,Z 459.858,A -85,B 0,C 180,E1 -8901.556,E2 -8901.556} C_VEL
LIN {X 0,Y 447.985,Z 465.179,A -85,B 0,C 180,E1 -8902.281,E2 -8902.281} C_VEL
LIN {X 0,Y 447.218,Z 469.084,A -85,B 0,C 180,E1 -8902.84,E2 -8902.84} C_VEL
LIN {X 0,Y 444.06,Z 475.187,A -85,B 0,C 180,E1 -8903.762,E2 -8903.762} C_VEL
LIN {X 0,Y 440.843,Z 480.62,A -85,B 0,C 180,E1 -8904.755,E2 -8904.755} C_VEL
LIN {X 0,Y 439.998,Z 483.475,A -85,B 0,C 180,E1 -8905.42,E2 -8905.42} C_VEL
LIN {X 0,Y 439.63,Z 488.335,A -85,B 0,C 180,E1 -8906.793,E2 -8906.793} C_VEL
LIN {X 0,Y 439.435,Z 492.087,A -85,B 0,C 180,E1 -8908.167,E2 -8908.167} C_VEL
LIN {X 0,Y 439.229,Z 495.559,A -85,B 0,C 180,E1 -8910,E2 -8910} C_VEL
LIN {X 0,Y 439.07,Z 496.71,A -85,B 0,C 180,E1 -8910.917,E2 -8910.917} C_VEL
LIN {X 0,Y 439.14,Z 497.406,A -85,B 0,C 180,E1 -8911.834,E2 -8911.834} C_VEL
LIN {X 0,Y 439.084,Z 497.724,A -85,B 0,C 180,E1 -8913.671,E2 -8913.671} C_VEL
LIN {X 0,Y 439.151,Z 497.311,A -85,B 0,C 180,E1 -8914.59,E2 -8914.59} C_VEL
LIN {X 0,Y 439.302,Z 496.466,A -85,B 0,C 180,E1 -8915.508,E2 -8915.508} C_VEL
LIN {X 0,Y 439.479,Z 493.643,A -85,B 0,C 180,E1 -8917.35,E2 -8917.35} C_VEL
LIN {X 0,Y 439.651,Z 490.403,A -85,B 0,C 180,E1 -8918.735,E2 -8918.735} C_VEL
LIN {X 0,Y 440.027,Z 486.086,A -85,B 0,C 180,E1 -8920.119,E2 -8920.119} C_VEL
LIN {X 0,Y 440.396,Z 480.593,A -85,B 0,C 180,E1 -8921.507,E2 -8921.507} C_VEL
LIN {X 0,Y 440.742,Z 473.69,A -85,B 0,C 180,E1 -8922.9,E2 -8922.9} C_VEL
LIN {X 0,Y 441.414,Z 465.005,A -85,B 0,C 180,E1 -8924.288,E2 -8924.288} C_VEL
LIN {X 0,Y 441.947,Z 456.079,A -85,B 0,C 180,E1 -8925.448,E2 -8925.448} C_VEL
LIN {X 0,Y 442.487,Z 446.165,A -85,B 0,C 180,E1 -8926.494,E2 -8926.494} C_VEL
LIN {X 0,Y 443.02,Z 435.085,A -85,B 0,C 180,E1 -8927.424,E2 -8927.424} C_VEL
LIN {X 0,Y 443.266,Z 430.179,A -85,B 0,C 180,E1 -8927.769,E2 -8927.769} C_VEL
LIN {X 0,Y 440.819,Z 421.157,A -85,B 0,C 180,E1 -8928.442,E2 -8928.442} C_VEL
LIN {X 0,Y 439.465,Z 416.746,A -85,B 0,C 180,E1 -8928.745,E2 -8928.745} C_VEL
LIN {X 0,Y 439.394,Z 416.752,A -85,B 0,C 180,E1 -8931.92,E2 -8931.92} C_VEL
LIN {X 0,Y 439.415,Z 416.75,A -85,B 0,C 180,E1 -8934.573,E2 -8934.573} C_VEL
LIN {X 0,Y 439.445,Z 416.742,A -85,B 0,C 180,E1 -8937.633,E2 -8937.633} C_VEL
LIN {X 0,Y 439.366,Z 416.753,A -85,B 0,C 180,E1 -8940.788,E2 -8940.788} C_VEL
LIN {X 0,Y 439.393,Z 416.754,A -85,B 0,C 180,E1 -8944.044,E2 -8944.044} C_VEL
LIN {X 0,Y 439.354,Z 416.753,A -85,B 0,C 180,E1 -8946.887,E2 -8946.887} C_VEL
LIN {X 0,Y 439.406,Z 416.75,A -85,B 0,C 180,E1 -8949.849,E2 -8949.849} C_VEL
LIN {X 0,Y 439.386,Z 416.75,A -85,B 0,C 180,E1 -8952.627,E2 -8952.627} C_VEL
LIN {X 0,Y 439.408,Z 416.746,A -85,B 0,C 180,E1 -8955.271,E2 -8955.271} C_VEL
LIN {X 0,Y 439.393,Z 416.748,A -85,B 0,C 180,E1 -8958.743,E2 -8958.743} C_VEL
LIN {X 0,Y 439.378,Z 416.753,A -85,B 0,C 180,E1 -8961.608,E2 -8961.608} C_VEL
LIN {X 0,Y 439.403,Z 416.747,A -85,B 0,C 180,E1 -8964.844,E2 -8964.844} C_VEL
LIN {X 0,Y 439.377,Z 416.755,A -85,B 0,C 180,E1 -8968.14,E2 -8968.14} C_VEL
LIN {X 0,Y 439.437,Z 416.747,A -85,B 0,C 180,E1 -8971.598,E2 -8971.598} C_VEL
LIN {X 0,Y 439.402,Z 416.748,A -85,B 0,C 180,E1 -8974.415,E2 -8974.415} C_VEL
LIN {X 0,Y 439.369,Z 416.754,A -85,B 0,C 180,E1 -8977.424,E2 -8977.424} C_VEL
LIN {X 0,Y 439.445,Z 416.741,A -85,B 0,C 180,E1 -8980.663,E2 -8980.663} C_VEL
LIN {X 0,Y 439.467,Z 416.741,A -85,B 0,C 180,E1 -8984.224,E2 -8984.224} C_VEL
LIN {X 0,Y 439.46,Z 416.747,A -85,B 0,C 180,E1 -8985.884,E2 -8985.884} C_VEL
LIN {X 0,Y 442.367,Z 428.135,A -85,B 0,C 180,E1 -8986.679,E2 -8986.679} C_VEL
LIN {X 0,Y 441.912,Z 437.518,A -85,B 0,C 180,E1 -8987.369,E2 -8987.369} C_VEL
LIN {X 0,Y 441.391,Z 448.824,A -85,B 0,C 180,E1 -8988.403,E2 -8988.403} C_VEL
LIN {X 0,Y 441.063,Z 458.046,A -85,B 0,C 180,E1 -8989.441,E2 -8989.441} C_VEL
LIN {X 0,Y 440.568,Z 466.552,A -85,B 0,C 180,E1 -8990.589,E2 -8990.589} C_VEL
LIN {X 0,Y 440.11,Z 475.051,A -85,B 0,C 180,E1 -8992.01,E2 -8992.01} C_VEL
LIN {X 0,Y 439.774,Z 481.516,A -85,B 0,C 180,E1 -8993.346,E2 -8993.346} C_VEL
LIN {X 0,Y 439.5,Z 487.638,A -85,B 0,C 180,E1 -8994.954,E2 -8994.954} C_VEL
LIN {X 0,Y 439.228,Z 491.64,A -85,B 0,C 180,E1 -8996.33,E2 -8996.33} C_VEL
LIN {X 0,Y 439.097,Z 493.722,A -85,B 0,C 180,E1 -8997.248,E2 -8997.248} C_VEL
LIN {X 0,Y 439.155,Z 495.371,A -85,B 0,C 180,E1 -8998.166,E2 -8998.166} C_VEL
LIN {X 0,Y 439.07,Z 496.596,A -85,B 0,C 180,E1 -8999.083,E2 -8999.083} C_VEL
LIN {X 0,Y 439.093,Z 497.823,A -85,B 0,C 180,E1 -9000.917,E2 -9000.917} C_VEL
LIN {X 0,Y 439.151,Z 497.845,A -85,B 0,C 180,E1 -9001.834,E2 -9001.834} C_VEL
LIN {X 0,Y 439.211,Z 496.647,A -85,B 0,C 180,E1 -9003.67,E2 -9003.67} C_VEL
LIN {X 0,Y 439.317,Z 495.462,A -85,B 0,C 180,E1 -9004.588,E2 -9004.588} C_VEL
LIN {X 0,Y 439.59,Z 492.839,A -85,B 0,C 180,E1 -9005.965,E2 -9005.965} C_VEL
LIN {X 0,Y 439.916,Z 488.594,A -85,B 0,C 180,E1 -9007.53,E2 -9007.53} C_VEL
LIN {X 0,Y 440.303,Z 482.532,A -85,B 0,C 180,E1 -9009.185,E2 -9009.185} C_VEL
LIN {X 0,Y 440.724,Z 475.964,A -85,B 0,C 180,E1 -9010.567,E2 -9010.567} C_VEL
LIN {X 0,Y 441.322,Z 467.709,A -85,B 0,C 180,E1 -9011.948,E2 -9011.948} C_VEL
LIN {X 0,Y 441.817,Z 459.287,A -85,B 0,C 180,E1 -9013.101,E2 -9013.101} C_VEL
LIN {X 0,Y 442.308,Z 450.251,A -85,B 0,C 180,E1 -9014.118,E2 -9014.118} C_VEL
LIN {X 0,Y 442.99,Z 438.464,A -85,B 0,C 180,E1 -9015.175,E2 -9015.175} C_VEL
LIN {X 0,Y 443.266,Z 429.133,A -85,B 0,C 180,E1 -9015.855,E2 -9015.855} C_VEL
LIN {X 0,Y 440.098,Z 418.934,A -85,B 0,C 180,E1 -9016.633,E2 -9016.633} C_VEL
LIN {X 0,Y 439.45,Z 416.748,A -85,B 0,C 180,E1 -9016.79,E2 -9016.79} C_VEL
LIN {X 0,Y 439.406,Z 416.758,A -85,B 0,C 180,E1 -9019.626,E2 -9019.626} C_VEL
LIN {X 0,Y 439.368,Z 416.759,A -85,B 0,C 180,E1 -9022.575,E2 -9022.575} C_VEL
LIN {X 0,Y 439.401,Z 416.754,A -85,B 0,C 180,E1 -9025.585,E2 -9025.585} C_VEL
LIN {X 0,Y 439.421,Z 416.752,A -85,B 0,C 180,E1 -9028.673,E2 -9028.673} C_VEL
LIN {X 0,Y 439.373,Z 416.755,A -85,B 0,C 180,E1 -9032.03,E2 -9032.03} C_VEL
LIN {X 0,Y 439.398,Z 416.752,A -85,B 0,C 180,E1 -9035.34,E2 -9035.34} C_VEL
LIN {X 0,Y 439.381,Z 416.755,A -85,B 0,C 180,E1 -9038.595,E2 -9038.595} C_VEL
LIN {X 0,Y 439.393,Z 416.75,A -85,B 0,C 180,E1 -9041.257,E2 -9041.257} C_VEL
LIN {X 0,Y 439.404,Z 416.753,A -85,B 0,C 180,E1 -9044.729,E2 -9044.729} C_VEL
LIN {X 0,Y 439.426,Z 416.803,A -85,B 0,C 180,E1 -9048.235,E2 -9048.235} C_VEL
LIN {X 0,Y 441.105,Z 425.154,A -85,B 0,C 180,E1 -9050.894,E2 -9050.894} C_VEL
LIN {X 0,Y 442.475,Z 432.637,A -85,B 0,C 180,E1 -9053.159,E2 -9053.159} C_VEL
LIN {X 0,Y 441.906,Z 441.11,A -85,B 0,C 180,E1 -9055.495,E2 -9055.495} C_VEL
LIN {X 0,Y 441.201,Z 453.653,A -85,B 0,C 180,E1 -9058.822,E2 -9058.822} C_VEL
LIN {X 0,Y 440.484,Z 467.761,A -85,B 0,C 180,E1 -9062.438,E2 -9062.438} C_VEL
LIN {X 0,Y 439.968,Z 480.27,A -85,B 0,C 180,E1 -9065.577,E2 -9065.577} C_VEL
LIN {X 0,Y 439.558,Z 491.769,A -85,B 0,C 180,E1 -9068.423,E2 -9068.423} C_VEL
LIN {X 0,Y 439.196,Z 505.524,A -85,B 0,C 180,E1 -9071.818,E2 -9071.818} C_VEL
LIN {X 0,Y 439.007,Z 512.175,A -85,B 0,C 180,E1 -9073.454,E2 -9073.454} C_VEL
LIN {X 0,Y 440.65,Z 527.218,A -85,B 0,C 180,E1 -9073.916,E2 -9073.916} C_VEL
LIN {X 0,Y 441.514,Z 540.043,A -85,B 0,C 180,E1 -9074.477,E2 -9074.477} C_VEL
LIN {X 0,Y 441.767,Z 546.678,A -85,B 0,C 180,E1 -9074.841,E2 -9074.841} C_VEL
LIN {X 0,Y 441.135,Z 558.289,A -85,B 0,C 180,E1 -9075.585,E2 -9075.585} C_VEL
LIN {X 0,Y 440.48,Z 569.588,A -85,B 0,C 180,E1 -9076.506,E2 -9076.506} C_VEL
LIN {X 0,Y 439.983,Z 579.803,A -85,B 0,C 180,E1 -9077.547,E2 -9077.547} C_VEL
LIN {X 0,Y 439.427,Z 589.06,A -85,B 0,C 180,E1 -9078.701,E2 -9078.701} C_VEL
LIN {X 0,Y 438.995,Z 598.133,A -85,B 0,C 180,E1 -9080.09,E2 -9080.09} C_VEL
LIN {X 0,Y 438.795,Z 605.469,A -85,B 0,C 180,E1 -9081.48,E2 -9081.48} C_VEL
LIN {X 0,Y 438.717,Z 612.186,A -85,B 0,C 180,E1 -9083.1,E2 -9083.1} C_VEL
LIN {X 0,Y 438.71,Z 616.641,A -85,B 0,C 180,E1 -9084.484,E2 -9084.484} C_VEL
LIN {X 0,Y 438.777,Z 619.016,A -85,B 0,C 180,E1 -9085.406,E2 -9085.406} C_VEL
LIN {X 0,Y 438.797,Z 620.931,A -85,B 0,C 180,E1 -9086.327,E2 -9086.327} C_VEL
LIN {X 0,Y 438.788,Z 622.365,A -85,B 0,C 180,E1 -9087.246,E2 -9087.246} C_VEL
LIN {X 0,Y 438.965,Z 624.043,A -85,B 0,C 180,E1 -9089.082,E2 -9089.082} C_VEL
LIN {X 0,Y 438.959,Z 624.256,A -85,B 0,C 180,E1 -9090,E2 -9090} C_VEL
LIN {X 0,Y 438.965,Z 624.027,A -85,B 0,C 180,E1 -9090.917,E2 -9090.917} C_VEL
LIN {X 0,Y 438.792,Z 622.336,A -85,B 0,C 180,E1 -9092.754,E2 -9092.754} C_VEL
LIN {X 0,Y 438.794,Z 620.878,A -85,B 0,C 180,E1 -9093.673,E2 -9093.673} C_VEL
LIN {X 0,Y 438.768,Z 617.825,A -85,B 0,C 180,E1 -9095.054,E2 -9095.054} C_VEL
LIN {X 0,Y 438.704,Z 612.87,A -85,B 0,C 180,E1 -9096.668,E2 -9096.668} C_VEL
LIN {X 0,Y 438.777,Z 606.294,A -85,B 0,C 180,E1 -9098.288,E2 -9098.288} C_VEL
LIN {X 0,Y 438.984,Z 599.159,A -85,B 0,C 180,E1 -9099.677,E2 -9099.677} C_VEL
LIN {X 0,Y 439.333,Z 590.238,A -85,B 0,C 180,E1 -9101.067,E2 -9101.067} C_VEL
LIN {X 0,Y 439.861,Z 581.143,A -85,B 0,C 180,E1 -9102.222,E2 -9102.222} C_VEL
LIN {X 0,Y 440.286,Z 571.643,A -85,B 0,C 180,E1 -9103.217,E2 -9103.217} C_VEL
LIN {X 0,Y 440.92,Z 560.206,A -85,B 0,C 180,E1 -9104.186,E2 -9104.186} C_VEL
LIN {X 0,Y 441.628,Z 547.962,A -85,B 0,C 180,E1 -9104.987,E2 -9104.987} C_VEL
LIN {X 0,Y 441.627,Z 542.587,A -85,B 0,C 180,E1 -9105.282,E2 -9105.282} C_VEL
LIN {X 0,Y 440.756,Z 531.612,A -85,B 0,C 180,E1 -9105.799,E2 -9105.799} C_VEL
LIN {X 0,Y 439.587,Z 518.306,A -85,B 0,C 180,E1 -9106.252,E2 -9106.252} C_VEL
LIN {X 0,Y 439.001,Z 512.46,A -85,B 0,C 180,E1 -9106.397,E2 -9106.397} C_VEL
LIN {X 0,Y 439.357,Z 499.208,A -85,B 0,C 180,E1 -9109.628,E2 -9109.628} C_VEL
LIN {X 0,Y 439.728,Z 485.208,A -85,B 0,C 180,E1 -9113.052,E2 -9113.052} C_VEL
LIN {X 0,Y 440.206,Z 472.01,A -85,B 0,C 180,E1 -9116.298,E2 -9116.298} C_VEL
LIN {X 0,Y 440.787,Z 458.717,A -85,B 0,C 180,E1 -9119.622,E2 -9119.622} C_VEL
LIN {X 0,Y 441.409,Z 445.375,A -85,B 0,C 180,E1 -9123.046,E2 -9123.046} C_VEL
LIN {X 0,Y 442.19,Z 433.103,A -85,B 0,C 180,E1 -9126.302,E2 -9126.302} C_VEL
LIN {X 0,Y 441.591,Z 427.833,A -85,B 0,C 180,E1 -9127.804,E2 -9127.804} C_VEL
LIN {X 0,Y 439.857,Z 418.84,A -85,B 0,C 180,E1 -9130.521,E2 -9130.521} C_VEL
LIN {X 0,Y 439.435,Z 416.75,A -85,B 0,C 180,E1 -9131.184,E2 -9131.184} C_VEL
LIN {X 0,Y 439.403,Z 416.758,A -85,B 0,C 180,E1 -9134.729,E2 -9134.729} C_VEL
LIN {X 0,Y 439.399,Z 416.752,A -85,B 0,C 180,E1 -9137.796,E2 -9137.796} C_VEL
LIN {X 0,Y 439.438,Z 416.75,A -85,B 0,C 180,E1 -9140.229,E2 -9140.229} C_VEL
LIN {X 0,Y 439.378,Z 416.755,A -85,B 0,C 180,E1 -9143.713,E2 -9143.713} C_VEL
LIN {X 0,Y 439.373,Z 416.753,A -85,B 0,C 180,E1 -9147.054,E2 -9147.054} C_VEL
LIN {X 0,Y 439.384,Z 416.756,A -85,B 0,C 180,E1 -9150.274,E2 -9150.274} C_VEL
LIN {X 0,Y 439.431,Z 416.747,A -85,B 0,C 180,E1 -9153.396,E2 -9153.396} C_VEL
LIN {X 0,Y 439.389,Z 416.755,A -85,B 0,C 180,E1 -9156.43,E2 -9156.43} C_VEL
LIN {X 0,Y 439.39,Z 416.752,A -85,B 0,C 180,E1 -9159.397,E2 -9159.397} C_VEL
LIN {X 0,Y 439.433,Z 416.75,A -85,B 0,C 180,E1 -9162.31,E2 -9162.31} C_VEL
LIN {X 0,Y 439.449,Z 416.744,A -85,B 0,C 180,E1 -9165.174,E2 -9165.174} C_VEL
LIN {X 0,Y 439.509,Z 416.74,A -85,B 0,C 180,E1 -9168.002,E2 -9168.002} C_VEL
LIN {X 0,Y 439.505,Z 416.74,A -85,B 0,C 180,E1 -9171.726,E2 -9171.726} C_VEL
LIN {X 0,Y 439.622,Z 416.725,A -85,B 0,C 180,E1 -9174.496,E2 -9174.496} C_VEL
LIN {X 0,Y 439.639,Z 416.724,A -85,B 0,C 180,E1 -9178.168,E2 -9178.168} C_VEL
LIN {X 0,Y 439.766,Z 416.709,A -85,B 0,C 180,E1 -9180,E2 -9180} C_VEL
LIN {X 0,Y 439.642,Z 416.72,A -85,B 0,C 180,E1 -9182.749,E2 -9182.749} C_VEL
LIN {X 0,Y 439.62,Z 416.726,A -85,B 0,C 180,E1 -9186.425,E2 -9186.425} C_VEL
LIN {X 0,Y 439.502,Z 416.738,A -85,B 0,C 180,E1 -9189.202,E2 -9189.202} C_VEL
LIN {X 0,Y 439.467,Z 416.742,A -85,B 0,C 180,E1 -9192.938,E2 -9192.938} C_VEL
LIN {X 0,Y 439.449,Z 416.747,A -85,B 0,C 180,E1 -9196.349,E2 -9196.349} C_VEL
LIN {X 0,Y 439.405,Z 416.752,A -85,B 0,C 180,E1 -9199.626,E2 -9199.626} C_VEL
LIN {X 0,Y 439.367,Z 416.756,A -85,B 0,C 180,E1 -9202.576,E2 -9202.576} C_VEL
LIN {X 0,Y 439.407,Z 416.753,A -85,B 0,C 180,E1 -9205.585,E2 -9205.585} C_VEL
LIN {X 0,Y 439.419,Z 416.748,A -85,B 0,C 180,E1 -9208.674,E2 -9208.674} C_VEL
LIN {X 0,Y 439.372,Z 416.757,A -85,B 0,C 180,E1 -9212.031,E2 -9212.031} C_VEL
LIN {X 0,Y 439.398,Z 416.753,A -85,B 0,C 180,E1 -9215.341,E2 -9215.341} C_VEL
LIN {X 0,Y 439.391,Z 416.752,A -85,B 0,C 180,E1 -9218.595,E2 -9218.595} C_VEL
LIN {X 0,Y 439.392,Z 416.752,A -85,B 0,C 180,E1 -9221.257,E2 -9221.257} C_VEL
LIN {X 0,Y 439.409,Z 416.749,A -85,B 0,C 180,E1 -9224.729,E2 -9224.729} C_VEL
LIN {X 0,Y 439.4,Z 416.755,A -85,B 0,C 180,E1 -9227.796,E2 -9227.796} C_VEL
LIN {X 0,Y 439.433,Z 416.748,A -85,B 0,C 180,E1 -9230.228,E2 -9230.228} C_VEL
LIN {X 0,Y 439.38,Z 416.757,A -85,B 0,C 180,E1 -9233.713,E2 -9233.713} C_VEL
LIN {X 0,Y 439.379,Z 416.754,A -85,B 0,C 180,E1 -9237.055,E2 -9237.055} C_VEL
LIN {X 0,Y 439.4,Z 416.752,A -85,B 0,C 180,E1 -9240.276,E2 -9240.276} C_VEL
LIN {X 0,Y 439.437,Z 416.749,A -85,B 0,C 180,E1 -9243.589,E2 -9243.589} C_VEL
LIN {X 0,Y 439.39,Z 416.752,A -85,B 0,C 180,E1 -9246.43,E2 -9246.43} C_VEL
LIN {X 0,Y 439.393,Z 416.754,A -85,B 0,C 180,E1 -9249.397,E2 -9249.397} C_VEL
LIN {X 0,Y 439.436,Z 416.747,A -85,B 0,C 180,E1 -9252.31,E2 -9252.31} C_VEL
LIN {X 0,Y 439.452,Z 416.747,A -85,B 0,C 180,E1 -9255.174,E2 -9255.174} C_VEL
LIN {X 0,Y 439.498,Z 416.74,A -85,B 0,C 180,E1 -9257.542,E2 -9257.542} C_VEL
LIN {X 0,Y 442.686,Z 428.019,A -85,B 0,C 180,E1 -9258.322,E2 -9258.322} C_VEL
LIN {X 0,Y 442.888,Z 431.415,A -85,B 0,C 180,E1 -9258.559,E2 -9258.559} C_VEL
LIN {X 0,Y 442.371,Z 443.068,A -85,B 0,C 180,E1 -9259.473,E2 -9259.473} C_VEL
LIN {X 0,Y 441.875,Z 453.58,A -85,B 0,C 180,E1 -9260.518,E2 -9260.518} C_VEL
LIN {X 0,Y 441.294,Z 462.312,A -85,B 0,C 180,E1 -9261.579,E2 -9261.579} C_VEL
LIN {X 0,Y 440.826,Z 471.124,A -85,B 0,C 180,E1 -9262.903,E2 -9262.903} C_VEL
LIN {X 0,Y 440.267,Z 478.471,A -85,B 0,C 180,E1 -9264.274,E2 -9264.274} C_VEL
LIN {X 0,Y 439.998,Z 483.475,A -85,B 0,C 180,E1 -9265.42,E2 -9265.42} C_VEL
LIN {X 0,Y 439.192,Z 486.152,A -85,B 0,C 180,E1 -9266.102,E2 -9266.102} C_VEL
LIN {X 0,Y 436.115,Z 490.258,A -85,B 0,C 180,E1 -9267.215,E2 -9267.215} C_VEL
LIN {X 0,Y 433.051,Z 493.673,A -85,B 0,C 180,E1 -9268.377,E2 -9268.377} C_VEL
LIN {X 0,Y 432.278,Z 495.194,A -85,B 0,C 180,E1 -9269.127,E2 -9269.127} C_VEL
LIN {X 0,Y 432.212,Z 496.621,A -85,B 0,C 180,E1 -9270,E2 -9270} C_VEL
LIN {X 0,Y 432.049,Z 497.751,A -85,B 0,C 180,E1 -9270.932,E2 -9270.932} C_VEL
LIN {X 0,Y 432.119,Z 498.434,A -85,B 0,C 180,E1 -9271.864,E2 -9271.864} C_VEL
LIN {X 0,Y 432.061,Z 498.731,A -85,B 0,C 180,E1 -9273.731,E2 -9273.731} C_VEL
LIN {X 0,Y 432.136,Z 498.299,A -85,B 0,C 180,E1 -9274.664,E2 -9274.664} C_VEL
LIN {X 0,Y 432.3,Z 497.438,A -85,B 0,C 180,E1 -9275.598,E2 -9275.598} C_VEL
LIN {X 0,Y 432.51,Z 494.591,A -85,B 0,C 180,E1 -9277.47,E2 -9277.47} C_VEL
LIN {X 0,Y 432.693,Z 491.327,A -85,B 0,C 180,E1 -9278.877,E2 -9278.877} C_VEL
LIN {X 0,Y 433.097,Z 486.984,A -85,B 0,C 180,E1 -9280.283,E2 -9280.283} C_VEL
LIN {X 0,Y 433.542,Z 480.387,A -85,B 0,C 180,E1 -9281.928,E2 -9281.928} C_VEL
LIN {X 0,Y 433.966,Z 473.383,A -85,B 0,C 180,E1 -9283.307,E2 -9283.307} C_VEL
LIN {X 0,Y 434.587,Z 465.787,A -85,B 0,C 180,E1 -9284.517,E2 -9284.517} C_VEL
LIN {X 0,Y 435.142,Z 456.817,A -85,B 0,C 180,E1 -9285.696,E2 -9285.696} C_VEL
LIN {X 0,Y 435.717,Z 446.813,A -85,B 0,C 180,E1 -9286.758,E2 -9286.758} C_VEL
LIN {X 0,Y 436.286,Z 435.534,A -85,B 0,C 180,E1 -9287.71,E2 -9287.71} C_VEL
LIN {X 0,Y 436.489,Z 431.548,A -85,B 0,C 180,E1 -9287.995,E2 -9287.995} C_VEL
LIN {X 0,Y 433.826,Z 422.205,A -85,B 0,C 180,E1 -9288.715,E2 -9288.715} C_VEL
LIN {X 0,Y 432.42,Z 417.622,A -85,B 0,C 180,E1 -9289.033,E2 -9289.033} C_VEL
LIN {X 0,Y 432.349,Z 417.631,A -85,B 0,C 180,E1 -9292.095,E2 -9292.095} C_VEL
LIN {X 0,Y 432.351,Z 417.626,A -85,B 0,C 180,E1 -9295.002,E2 -9295.002} C_VEL
LIN {X 0,Y 432.386,Z 417.626,A -85,B 0,C 180,E1 -9298.123,E2 -9298.123} C_VEL
LIN {X 0,Y 432.326,Z 417.628,A -85,B 0,C 180,E1 -9301.346,E2 -9301.346} C_VEL
LIN {X 0,Y 432.346,Z 417.628,A -85,B 0,C 180,E1 -9304.677,E2 -9304.677} C_VEL
LIN {X 0,Y 432.342,Z 417.634,A -85,B 0,C 180,E1 -9308.15,E2 -9308.15} C_VEL
LIN {X 0,Y 432.337,Z 417.629,A -85,B 0,C 180,E1 -9311.602,E2 -9311.602} C_VEL
LIN {X 0,Y 432.338,Z 417.631,A -85,B 0,C 180,E1 -9314.347,E2 -9314.347} C_VEL
LIN {X 0,Y 432.325,Z 417.628,A -85,B 0,C 180,E1 -9317.016,E2 -9317.016} C_VEL
LIN {X 0,Y 432.337,Z 417.632,A -85,B 0,C 180,E1 -9319.821,E2 -9319.821} C_VEL
LIN {X 0,Y 432.311,Z 417.63,A -85,B 0,C 180,E1 -9323.022,E2 -9323.022} C_VEL
LIN {X 0,Y 432.364,Z 417.631,A -85,B 0,C 180,E1 -9325.996,E2 -9325.996} C_VEL
LIN {X 0,Y 432.352,Z 417.628,A -85,B 0,C 180,E1 -9329.49,E2 -9329.49} C_VEL
LIN {X 0,Y 432.395,Z 417.62,A -85,B 0,C 180,E1 -9332.928,E2 -9332.928} C_VEL
LIN {X 0,Y 432.372,Z 417.627,A -85,B 0,C 180,E1 -9336.023,E2 -9336.023} C_VEL
LIN {X 0,Y 432.354,Z 417.625,A -85,B 0,C 180,E1 -9339.046,E2 -9339.046} C_VEL
LIN {X 0,Y 432.378,Z 417.626,A -85,B 0,C 180,E1 -9342.011,E2 -9342.011} C_VEL
LIN {X 0,Y 432.4,Z 417.619,A -85,B 0,C 180,E1 -9344.926,E2 -9344.926} C_VEL
LIN {X 0,Y 432.441,Z 417.816,A -85,B 0,C 180,E1 -9345.695,E2 -9345.695} C_VEL
LIN {X 0,Y 435.452,Z 429.274,A -85,B 0,C 180,E1 -9346.509,E2 -9346.509} C_VEL
LIN {X 0,Y 435.002,Z 439.436,A -85,B 0,C 180,E1 -9347.283,E2 -9347.283} C_VEL
LIN {X 0,Y 434.408,Z 450.58,A -85,B 0,C 180,E1 -9348.332,E2 -9348.332} C_VEL
LIN {X 0,Y 434.006,Z 460.573,A -85,B 0,C 180,E1 -9349.503,E2 -9349.503} C_VEL
LIN {X 0,Y 433.434,Z 470.257,A -85,B 0,C 180,E1 -9350.904,E2 -9350.904} C_VEL
LIN {X 0,Y 433.092,Z 477.346,A -85,B 0,C 180,E1 -9352.166,E2 -9352.166} C_VEL
LIN {X 0,Y 432.709,Z 483.366,A -85,B 0,C 180,E1 -9353.472,E2 -9353.472} C_VEL
LIN {X 0,Y 432.5,Z 488.531,A -85,B 0,C 180,E1 -9354.872,E2 -9354.872} C_VEL
LIN {X 0,Y 432.205,Z 492.573,A -85,B 0,C 180,E1 -9356.27,E2 -9356.27} C_VEL
LIN {X 0,Y 432.07,Z 494.672,A -85,B 0,C 180,E1 -9357.203,E2 -9357.203} C_VEL
LIN {X 0,Y 432.135,Z 496.344,A -85,B 0,C 180,E1 -9358.136,E2 -9358.136} C_VEL
LIN {X 0,Y 432.048,Z 497.599,A -85,B 0,C 180,E1 -9359.068,E2 -9359.068} C_VEL
LIN {X 0,Y 432.094,Z 498.862,A -85,B 0,C 180,E1 -9360.932,E2 -9360.932} C_VEL
LIN {X 0,Y 432.161,Z 498.907,A -85,B 0,C 180,E1 -9361.864,E2 -9361.864} C_VEL
LIN {X 0,Y 432.209,Z 497.746,A -85,B 0,C 180,E1 -9363.729,E2 -9363.729} C_VEL
LIN {X 0,Y 432.325,Z 496.576,A -85,B 0,C 180,E1 -9364.662,E2 -9364.662} C_VEL
LIN {X 0,Y 432.631,Z 493.969,A -85,B 0,C 180,E1 -9366.061,E2 -9366.061} C_VEL
LIN {X 0,Y 432.999,Z 489.59,A -85,B 0,C 180,E1 -9367.7,E2 -9367.7} C_VEL
LIN {X 0,Y 433.416,Z 483.704,A -85,B 0,C 180,E1 -9369.332,E2 -9369.332} C_VEL
LIN {X 0,Y 433.87,Z 477.196,A -85,B 0,C 180,E1 -9370.736,E2 -9370.736} C_VEL
LIN {X 0,Y 434.51,Z 469.016,A -85,B 0,C 180,E1 -9372.138,E2 -9372.138} C_VEL
LIN {X 0,Y 435.047,Z 460.648,A -85,B 0,C 180,E1 -9373.309,E2 -9373.309} C_VEL
LIN {X 0,Y 435.597,Z 451.365,A -85,B 0,C 180,E1 -9374.37,E2 -9374.37} C_VEL
LIN {X 0,Y 436.28,Z 439.947,A -85,B 0,C 180,E1 -9375.414,E2 -9375.414} C_VEL
LIN {X 0,Y 436.47,Z 430.307,A -85,B 0,C 180,E1 -9376.138,E2 -9376.138} C_VEL
LIN {X 0,Y 433.012,Z 419.733,A -85,B 0,C 180,E1 -9376.987,E2 -9376.987} C_VEL
LIN {X 0,Y 432.396,Z 417.629,A -85,B 0,C 180,E1 -9377.133,E2 -9377.133} C_VEL
LIN {X 0,Y 432.343,Z 417.638,A -85,B 0,C 180,E1 -9379.96,E2 -9379.96} C_VEL
LIN {X 0,Y 432.321,Z 417.636,A -85,B 0,C 180,E1 -9382.964,E2 -9382.964} C_VEL
LIN {X 0,Y 432.364,Z 417.628,A -85,B 0,C 180,E1 -9386.032,E2 -9386.032} C_VEL
LIN {X 0,Y 432.347,Z 417.631,A -85,B 0,C 180,E1 -9389.187,E2 -9389.187} C_VEL
LIN {X 0,Y 432.326,Z 417.634,A -85,B 0,C 180,E1 -9392.443,E2 -9392.443} C_VEL
LIN {X 0,Y 432.347,Z 417.63,A -85,B 0,C 180,E1 -9395.632,E2 -9395.632} C_VEL
LIN {X 0,Y 432.349,Z 417.629,A -85,B 0,C 180,E1 -9399.343,E2 -9399.343} C_VEL
LIN {X 0,Y 432.338,Z 417.628,A -85,B 0,C 180,E1 -9401.797,E2 -9401.797} C_VEL
LIN {X 0,Y 432.336,Z 417.631,A -85,B 0,C 180,E1 -9404.347,E2 -9404.347} C_VEL
LIN {X 0,Y 432.373,Z 417.703,A -85,B 0,C 180,E1 -9407.894,E2 -9407.894} C_VEL
LIN {X 0,Y 434.274,Z 427.123,A -85,B 0,C 180,E1 -9410.969,E2 -9410.969} C_VEL
LIN {X 0,Y 435.448,Z 433.248,A -85,B 0,C 180,E1 -9412.847,E2 -9412.847} C_VEL
LIN {X 0,Y 435.208,Z 438.878,A -85,B 0,C 180,E1 -9414.454,E2 -9414.454} C_VEL
LIN {X 0,Y 434.334,Z 451.88,A -85,B 0,C 180,E1 -9417.999,E2 -9417.999} C_VEL
LIN {X 0,Y 433.734,Z 463.428,A -85,B 0,C 180,E1 -9421.044,E2 -9421.044} C_VEL
LIN {X 0,Y 433.162,Z 474.964,A -85,B 0,C 180,E1 -9424.019,E2 -9424.019} C_VEL
LIN {X 0,Y 432.65,Z 488.643,A -85,B 0,C 180,E1 -9427.492,E2 -9427.492} C_VEL
LIN {X 0,Y 432.191,Z 502.649,A -85,B 0,C 180,E1 -9431.02,E2 -9431.02} C_VEL
LIN {X 0,Y 431.932,Z 511.105,A -85,B 0,C 180,E1 -9433.151,E2 -9433.151} C_VEL
LIN {X 0,Y 433.686,Z 526.719,A -85,B 0,C 180,E1 -9433.652,E2 -9433.652} C_VEL
LIN {X 0,Y 434.541,Z 540.447,A -85,B 0,C 180,E1 -9434.282,E2 -9434.282} C_VEL
LIN {X 0,Y 434.835,Z 546.912,A -85,B 0,C 180,E1 -9434.653,E2 -9434.653} C_VEL
LIN {X 0,Y 434.122,Z 559.059,A -85,B 0,C 180,E1 -9435.467,E2 -9435.467} C_VEL
LIN {X 0,Y 433.419,Z 570.412,A -85,B 0,C 180,E1 -9436.449,E2 -9436.449} C_VEL
LIN {X 0,Y 432.963,Z 578.937,A -85,B 0,C 180,E1 -9437.347,E2 -9437.347} C_VEL
LIN {X 0,Y 432.407,Z 588.129,A -85,B 0,C 180,E1 -9438.515,E2 -9438.515} C_VEL
LIN {X 0,Y 431.926,Z 597.181,A -85,B 0,C 180,E1 -9439.926,E2 -9439.926} C_VEL
LIN {X 0,Y 431.718,Z 604.499,A -85,B 0,C 180,E1 -9441.339,E2 -9441.339} C_VEL
LIN {X 0,Y 431.638,Z 609.468,A -85,B 0,C 180,E1 -9442.515,E2 -9442.515} C_VEL
LIN {X 0,Y 431.676,Z 614.316,A -85,B 0,C 180,E1 -9443.925,E2 -9443.925} C_VEL
LIN {X 0,Y 431.733,Z 618.026,A -85,B 0,C 180,E1 -9445.331,E2 -9445.331} C_VEL
LIN {X 0,Y 431.757,Z 619.935,A -85,B 0,C 180,E1 -9446.267,E2 -9446.267} C_VEL
LIN {X 0,Y 431.744,Z 621.364,A -85,B 0,C 180,E1 -9447.201,E2 -9447.201} C_VEL
LIN {X 0,Y 431.944,Z 623.038,A -85,B 0,C 180,E1 -9449.068,E2 -9449.068} C_VEL
LIN {X 0,Y 431.941,Z 623.244,A -85,B 0,C 180,E1 -9450,E2 -9450} C_VEL
LIN {X 0,Y 431.944,Z 623.009,A -85,B 0,C 180,E1 -9450.932,E2 -9450.932} C_VEL
LIN {X 0,Y 431.751,Z 621.305,A -85,B 0,C 180,E1 -9452.799,E2 -9452.799} C_VEL
LIN {X 0,Y 431.754,Z 619.839,A -85,B 0,C 180,E1 -9453.733,E2 -9453.733} C_VEL
LIN {X 0,Y 431.719,Z 616.775,A -85,B 0,C 180,E1 -9455.137,E2 -9455.137} C_VEL
LIN {X 0,Y 431.641,Z 612.14,A -85,B 0,C 180,E1 -9456.682,E2 -9456.682} C_VEL
LIN {X 0,Y 431.702,Z 606.251,A -85,B 0,C 180,E1 -9458.189,E2 -9458.189} C_VEL
LIN {X 0,Y 431.88,Z 599.328,A -85,B 0,C 180,E1 -9459.602,E2 -9459.602} C_VEL
LIN {X 0,Y 432.24,Z 590.766,A -85,B 0,C 180,E1 -9461.014,E2 -9461.014} C_VEL
LIN {X 0,Y 432.716,Z 581.978,A -85,B 0,C 180,E1 -9462.189,E2 -9462.189} C_VEL
LIN {X 0,Y 433.125,Z 572.846,A -85,B 0,C 180,E1 -9463.2,E2 -9463.2} C_VEL
LIN {X 0,Y 433.812,Z 561.926,A -85,B 0,C 180,E1 -9464.184,E2 -9464.184} C_VEL
LIN {X 0,Y 434.481,Z 550.544,A -85,B 0,C 180,E1 -9464.999,E2 -9464.999} C_VEL
LIN {X 0,Y 434.673,Z 543.552,A -85,B 0,C 180,E1 -9465.413,E2 -9465.413} C_VEL
LIN {X 0,Y 433.888,Z 533.523,A -85,B 0,C 180,E1 -9465.923,E2 -9465.923} C_VEL
LIN {X 0,Y 432.802,Z 520.233,A -85,B 0,C 180,E1 -9466.421,E2 -9466.421} C_VEL
LIN {X 0,Y 431.922,Z 511.387,A -85,B 0,C 180,E1 -9466.668,E2 -9466.668} C_VEL
LIN {X 0,Y 432.283,Z 498.165,A -85,B 0,C 180,E1 -9469.963,E2 -9469.963} C_VEL
LIN {X 0,Y 432.684,Z 485.218,A -85,B 0,C 180,E1 -9473.197,E2 -9473.197} C_VEL
LIN {X 0,Y 433.174,Z 472.411,A -85,B 0,C 180,E1 -9476.409,E2 -9476.409} C_VEL
LIN {X 0,Y 433.865,Z 457.789,A -85,B 0,C 180,E1 -9480.143,E2 -9480.143} C_VEL
LIN {X 0,Y 434.515,Z 444.481,A -85,B 0,C 180,E1 -9483.64,E2 -9483.64} C_VEL
LIN {X 0,Y 435.224,Z 433.249,A -85,B 0,C 180,E1 -9486.689,E2 -9486.689} C_VEL
LIN {X 0,Y 433.81,Z 424.887,A -85,B 0,C 180,E1 -9489.185,E2 -9489.185} C_VEL
LIN {X 0,Y 432.366,Z 417.631,A -85,B 0,C 180,E1 -9491.488,E2 -9491.488} C_VEL
LIN {X 0,Y 432.334,Z 417.637,A -85,B 0,C 180,E1 -9494.347,E2 -9494.347} C_VEL
